Yaskawa INFORM job: A_ROOF_SIDE_0617_2_PAINT_25.JBI

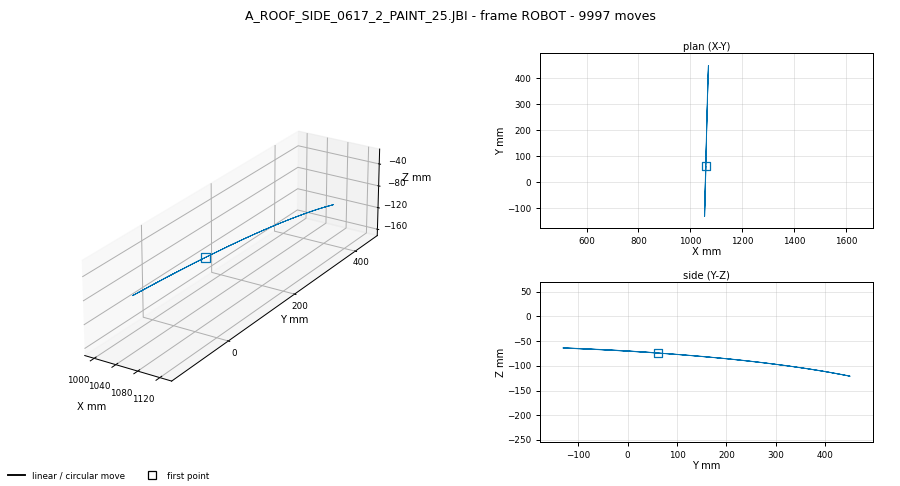
[picture p0: tool path of A_ROOF_SIDE_0617_2_PAINT_25.JBI in frame ROBOT, 9997 of 9997 moves have a stored position in this frame; points joined in program order, loops and branches not executed]
/JOB
//NAME A_ROOF_SIDE_0617_2_PAINT25
//POS
///NPOS 9997,0,0,0,0,0
///TOOL 1
///USER 0
///POSTYPE ROBOT
///RECTAN
///RCONF 1,0,0,0,0,0,0,0,0,0,0,0,0,0,0,0,0,0,0,0,0,0,0,0
C00000=1059.845,61.842,-73.709,171.756,29.525,155.487
C00001=1059.838,61.557,-73.690,171.754,29.522,155.486
C00002=1059.832,61.309,-73.673,171.753,29.519,155.486
C00003=1059.826,61.059,-73.655,171.752,29.517,155.485
C00004=1059.820,60.810,-73.638,171.750,29.515,155.485
C00005=1059.814,60.561,-73.621,171.748,29.512,155.485
C00006=1059.807,60.311,-73.604,171.747,29.509,155.484
C00007=1059.801,60.062,-73.587,171.746,29.507,155.484
C00008=1059.795,59.813,-73.569,171.744,29.505,155.484
C00009=1059.789,59.563,-73.553,171.743,29.502,155.483
C00010=1059.783,59.314,-73.535,171.741,29.500,155.483
C00011=1059.777,59.065,-73.518,171.739,29.497,155.482
C00012=1059.771,58.816,-73.501,171.739,29.494,155.482
C00013=1059.765,58.566,-73.483,171.737,29.492,155.482
C00014=1059.758,58.317,-73.466,171.735,29.489,155.481
C00015=1059.752,58.067,-73.450,171.733,29.487,155.481
C00016=1059.746,57.818,-73.432,171.733,29.485,155.481
C00017=1059.740,57.569,-73.415,171.731,29.482,155.480
C00018=1059.734,57.319,-73.398,171.729,29.479,155.480
C00019=1059.728,57.070,-73.381,171.728,29.477,155.480
C00020=1059.722,56.821,-73.365,171.726,29.474,155.479
C00021=1059.716,56.571,-73.347,171.725,29.472,155.479
C00022=1059.710,56.322,-73.330,171.723,29.470,155.478
C00023=1059.703,56.072,-73.313,171.722,29.467,155.478
C00024=1059.698,55.823,-73.296,171.720,29.464,155.478
C00025=1059.692,55.574,-73.279,171.719,29.462,155.477
C00026=1059.685,55.324,-73.262,171.718,29.459,155.477
C00027=1059.680,55.075,-73.245,171.716,29.457,155.477
C00028=1059.673,54.826,-73.228,171.714,29.454,155.476
C00029=1059.666,54.577,-73.211,171.712,29.452,155.476
C00030=1059.661,54.327,-73.194,171.712,29.449,155.475
C00031=1059.655,54.078,-73.177,171.710,29.446,155.475
C00032=1059.648,53.828,-73.161,171.708,29.444,155.475
C00033=1059.643,53.579,-73.143,171.707,29.441,155.474
C00034=1059.637,53.330,-73.127,171.706,29.439,155.474
C00035=1059.631,53.081,-73.110,171.704,29.437,155.474
C00036=1059.625,52.831,-73.093,171.703,29.434,155.473
C00037=1059.619,52.582,-73.076,171.701,29.431,155.473
C00038=1059.613,52.333,-73.059,171.700,29.429,155.473
C00039=1059.607,52.083,-73.041,171.698,29.426,155.472
C00040=1059.601,51.834,-73.025,171.697,29.424,155.472
C00041=1059.595,51.584,-73.009,171.695,29.422,155.472
C00042=1059.589,51.335,-72.991,171.693,29.419,155.471
C00043=1059.583,51.085,-72.975,171.693,29.416,155.471
C00044=1059.576,50.836,-72.958,171.691,29.413,155.470
C00045=1059.571,50.587,-72.941,171.689,29.411,155.470
C00046=1059.565,50.338,-72.924,171.688,29.409,155.470
C00047=1059.558,50.088,-72.907,171.687,29.406,155.469
C00048=1059.553,49.838,-72.890,171.685,29.404,155.469
C00049=1059.547,49.590,-72.873,171.683,29.401,155.469
C00050=1059.541,49.340,-72.857,171.682,29.398,155.468
C00051=1059.534,49.091,-72.840,171.680,29.396,155.468
C00052=1059.529,48.841,-72.823,171.679,29.394,155.467
C00053=1059.523,48.592,-72.807,171.678,29.391,155.467
C00054=1059.517,48.343,-72.790,171.676,29.388,155.467
C00055=1059.511,48.093,-72.773,171.674,29.386,155.466
C00056=1059.505,47.843,-72.756,171.674,29.383,155.466
C00057=1059.499,47.595,-72.739,171.672,29.381,155.466
C00058=1059.493,47.345,-72.723,171.670,29.378,155.465
C00059=1059.487,47.096,-72.706,171.668,29.376,155.465
C00060=1059.481,46.847,-72.689,171.668,29.373,155.464
C00061=1059.475,46.597,-72.673,171.666,29.370,155.464
C00062=1059.468,46.313,-72.654,171.664,29.368,155.464
C00063=1059.462,46.027,-72.634,171.663,29.365,155.463
C00064=1059.455,45.742,-72.615,171.661,29.361,155.463
C00065=1059.448,45.458,-72.596,171.659,29.359,155.462
C00066=1059.442,45.208,-72.580,171.658,29.356,155.462
C00067=1059.436,44.959,-72.563,171.656,29.354,155.462
C00068=1059.430,44.709,-72.547,171.654,29.351,155.461
C00069=1059.424,44.461,-72.530,171.654,29.348,155.461
C00070=1059.419,44.211,-72.513,171.652,29.346,155.461
C00071=1059.412,43.961,-72.497,171.650,29.343,155.460
C00072=1059.406,43.711,-72.480,171.649,29.341,155.460
C00073=1059.401,43.462,-72.464,171.648,29.338,155.459
C00074=1059.394,43.213,-72.447,171.646,29.336,155.459
C00075=1059.388,42.964,-72.431,171.645,29.333,155.459
C00076=1059.382,42.715,-72.415,171.643,29.331,155.458
C00077=1059.376,42.465,-72.398,171.641,29.328,155.458
C00078=1059.370,42.215,-72.382,171.640,29.326,155.458
C00079=1059.364,41.966,-72.365,171.639,29.324,155.457
C00080=1059.358,41.717,-72.349,171.637,29.321,155.457
C00081=1059.352,41.468,-72.332,171.635,29.319,155.457
C00082=1059.346,41.218,-72.316,171.635,29.316,155.456
C00083=1059.340,40.969,-72.300,171.633,29.313,155.456
C00084=1059.333,40.719,-72.283,171.631,29.311,155.455
C00085=1059.327,40.470,-72.267,171.630,29.308,155.455
C00086=1059.322,40.220,-72.250,171.628,29.306,155.455
C00087=1059.316,39.971,-72.234,171.627,29.304,155.454
C00088=1059.310,39.721,-72.217,171.625,29.301,155.454
C00089=1059.304,39.472,-72.201,171.624,29.299,155.454
C00090=1059.298,39.223,-72.185,171.622,29.296,155.453
C00091=1059.292,38.973,-72.169,171.620,29.293,155.453
C00092=1059.286,38.724,-72.152,171.620,29.291,155.453
C00093=1059.280,38.474,-72.136,171.618,29.288,155.452
C00094=1059.274,38.225,-72.120,171.616,29.286,155.452
C00095=1059.268,37.975,-72.103,171.615,29.283,155.452
C00096=1059.262,37.726,-72.087,171.614,29.281,155.451
C00097=1059.255,37.477,-72.071,171.612,29.279,155.451
C00098=1059.249,37.228,-72.055,171.610,29.276,155.450
C00099=1059.243,36.978,-72.039,171.609,29.274,155.450
C00100=1059.237,36.729,-72.023,171.607,29.271,155.450
C00101=1059.231,36.479,-72.006,171.606,29.269,155.449
C00102=1059.224,36.230,-71.990,171.605,29.266,155.449
C00103=1059.218,35.980,-71.974,171.603,29.264,155.449
C00104=1059.212,35.731,-71.958,171.601,29.261,155.448
C00105=1059.206,35.482,-71.942,171.600,29.259,155.448
C00106=1059.200,35.232,-71.925,171.599,29.256,155.448
C00107=1059.194,34.983,-71.910,171.597,29.254,155.447
C00108=1059.188,34.734,-71.893,171.595,29.252,155.447
C00109=1059.182,34.484,-71.878,171.594,29.249,155.447
C00110=1059.176,34.235,-71.862,171.593,29.247,155.446
C00111=1059.170,33.985,-71.845,171.591,29.244,155.446
C00112=1059.164,33.736,-71.830,171.590,29.242,155.446
C00113=1059.158,33.487,-71.813,171.588,29.239,155.445
C00114=1059.152,33.238,-71.797,171.586,29.237,155.445
C00115=1059.146,32.988,-71.781,171.586,29.234,155.445
C00116=1059.139,32.738,-71.765,171.584,29.232,155.444
C00117=1059.133,32.488,-71.749,171.582,29.229,155.444
C00118=1059.127,32.239,-71.733,171.580,29.227,155.444
C00119=1059.121,31.990,-71.717,171.579,29.224,155.443
C00120=1059.115,31.740,-71.701,171.578,29.222,155.443
C00121=1059.108,31.491,-71.686,171.576,29.220,155.443
C00122=1059.103,31.241,-71.669,171.575,29.217,155.442
C00123=1059.097,30.992,-71.653,171.573,29.215,155.442
C00124=1059.091,30.743,-71.637,171.571,29.212,155.442
C00125=1059.085,30.493,-71.621,171.571,29.210,155.441
C00126=1059.078,30.209,-71.603,171.569,29.207,155.441
C00127=1059.071,29.923,-71.585,171.567,29.204,155.440
C00128=1059.064,29.639,-71.566,171.565,29.201,155.440
C00129=1059.057,29.354,-71.549,171.563,29.199,155.440
C00130=1059.051,29.105,-71.532,171.562,29.196,155.439
C00131=1059.045,28.855,-71.517,171.561,29.194,155.439
C00132=1059.039,28.606,-71.501,171.559,29.191,155.439
C00133=1059.033,28.356,-71.485,171.557,29.189,155.438
C00134=1059.027,28.106,-71.469,171.556,29.186,155.438
C00135=1059.020,27.857,-71.454,171.555,29.184,155.438
C00136=1059.014,27.608,-71.438,171.553,29.181,155.437
C00137=1059.009,27.358,-71.422,171.551,29.179,155.437
C00138=1059.002,27.109,-71.406,171.550,29.177,155.437
C00139=1058.996,26.860,-71.390,171.548,29.174,155.436
C00140=1058.990,26.610,-71.375,171.547,29.172,155.436
C00141=1058.984,26.361,-71.359,171.546,29.169,155.436
C00142=1058.977,26.111,-71.343,171.544,29.167,155.435
C00143=1058.971,25.862,-71.328,171.542,29.164,155.435
C00144=1058.965,25.612,-71.311,171.541,29.162,155.435
C00145=1058.959,25.363,-71.296,171.540,29.160,155.434
C00146=1058.953,25.113,-71.280,171.538,29.158,155.434
C00147=1058.946,24.864,-71.265,171.536,29.155,155.434
C00148=1058.941,24.614,-71.249,171.535,29.153,155.433
C00149=1058.935,24.366,-71.234,171.533,29.150,155.433
C00150=1058.929,24.116,-71.218,171.532,29.148,155.432
C00151=1058.922,23.867,-71.203,171.531,29.146,155.432
C00152=1058.917,23.617,-71.187,171.529,29.143,155.432
C00153=1058.910,23.368,-71.171,171.527,29.141,155.432
C00154=1058.904,23.118,-71.156,171.526,29.138,155.431
C00155=1058.898,22.869,-71.140,171.525,29.136,155.431
C00156=1058.892,22.619,-71.125,171.523,29.134,155.431
C00157=1058.886,22.369,-71.108,171.522,29.131,155.430
C00158=1058.880,22.120,-71.093,171.520,29.129,155.430
C00159=1058.874,21.870,-71.077,171.518,29.126,155.430
C00160=1058.868,21.622,-71.063,171.517,29.124,155.429
C00161=1058.862,21.372,-71.046,171.516,29.122,155.429
C00162=1058.856,21.123,-71.031,171.514,29.119,155.429
C00163=1058.850,20.873,-71.015,171.512,29.117,155.428
C00164=1058.843,20.624,-71.000,171.511,29.114,155.428
C00165=1058.837,20.374,-70.984,171.509,29.112,155.428
C00166=1058.831,20.125,-70.969,171.508,29.109,155.427
C00167=1058.825,19.875,-70.954,171.507,29.107,155.427
C00168=1058.819,19.626,-70.938,171.505,29.105,155.427
C00169=1058.813,19.377,-70.923,171.503,29.102,155.426
C00170=1058.807,19.127,-70.907,171.502,29.100,155.426
C00171=1058.801,18.878,-70.892,171.501,29.098,155.426
C00172=1058.794,18.628,-70.877,171.499,29.095,155.425
C00173=1058.788,18.379,-70.861,171.497,29.093,155.425
C00174=1058.782,18.129,-70.846,171.496,29.090,155.425
C00175=1058.776,17.879,-70.830,171.494,29.088,155.424
C00176=1058.770,17.631,-70.815,171.493,29.086,155.424
C00177=1058.764,17.381,-70.800,171.492,29.083,155.424
C00178=1058.758,17.131,-70.784,171.490,29.081,155.423
C00179=1058.751,16.882,-70.769,171.488,29.079,155.423
C00180=1058.745,16.632,-70.754,171.487,29.076,155.423
C00181=1058.739,16.382,-70.738,171.485,29.074,155.422
C00182=1058.733,16.134,-70.723,171.484,29.071,155.422
C00183=1058.728,15.884,-70.707,171.482,29.069,155.422
C00184=1058.721,15.634,-70.693,171.481,29.067,155.421
C00185=1058.715,15.385,-70.678,171.479,29.064,155.421
C00186=1058.709,15.135,-70.661,171.477,29.062,155.421
C00187=1058.703,14.886,-70.647,171.477,29.060,155.420
C00188=1058.697,14.637,-70.632,171.475,29.057,155.420
C00189=1058.691,14.387,-70.616,171.473,29.055,155.420
C00190=1058.684,14.104,-70.599,171.472,29.052,155.419
C00191=1058.676,13.820,-70.581,171.470,29.050,155.419
C00192=1058.669,13.537,-70.565,171.468,29.047,155.419
C00193=1058.662,13.253,-70.547,171.467,29.044,155.418
C00194=1058.656,13.004,-70.532,171.465,29.042,155.418
C00195=1058.650,12.754,-70.517,171.463,29.040,155.418
C00196=1058.644,12.504,-70.502,171.462,29.037,155.417
C00197=1058.637,12.255,-70.487,171.460,29.035,155.417
C00198=1058.631,12.005,-70.472,171.458,29.033,155.417
C00199=1058.625,11.756,-70.457,171.457,29.031,155.417
C00200=1058.619,11.507,-70.442,171.456,29.028,155.416
C00201=1058.613,11.257,-70.427,171.454,29.026,155.416
C00202=1058.606,11.007,-70.412,171.452,29.023,155.416
C00203=1058.600,10.758,-70.397,171.451,29.021,155.415
C00204=1058.594,10.509,-70.382,171.449,29.019,155.415
C00205=1058.588,10.259,-70.367,171.447,29.016,155.415
C00206=1058.581,10.010,-70.352,171.447,29.014,155.414
C00207=1058.576,9.760,-70.337,171.445,29.012,155.414
C00208=1058.570,9.511,-70.322,171.443,29.010,155.414
C00209=1058.563,9.262,-70.307,171.442,29.007,155.413
C00210=1058.557,9.012,-70.292,171.440,29.005,155.413
C00211=1058.551,8.762,-70.277,171.438,29.003,155.413
C00212=1058.545,8.513,-70.262,171.437,29.001,155.413
C00213=1058.538,8.264,-70.247,171.436,28.999,155.412
C00214=1058.532,8.014,-70.232,171.434,28.996,155.412
C00215=1058.526,7.764,-70.217,171.432,28.994,155.412
C00216=1058.520,7.515,-70.203,171.431,28.991,155.411
C00217=1058.514,7.265,-70.187,171.429,28.989,155.411
C00218=1058.508,7.016,-70.172,171.428,28.987,155.411
C00219=1058.502,6.767,-70.158,171.427,28.984,155.410
C00220=1058.496,6.517,-70.143,171.425,28.982,155.410
C00221=1058.489,6.267,-70.128,171.423,28.980,155.410
C00222=1058.483,6.018,-70.113,171.421,28.978,155.410
C00223=1058.477,5.769,-70.098,171.420,28.975,155.409
C00224=1058.471,5.519,-70.083,171.418,28.973,155.409
C00225=1058.464,5.270,-70.068,171.417,28.971,155.409
C00226=1058.459,5.020,-70.054,171.416,28.969,155.408
C00227=1058.452,4.770,-70.039,171.414,28.966,155.408
C00228=1058.446,4.521,-70.024,171.412,28.964,155.408
C00229=1058.440,4.272,-70.010,171.411,28.961,155.407
C00230=1058.434,4.022,-69.995,171.409,28.959,155.407
C00231=1058.428,3.772,-69.979,171.408,28.957,155.407
C00232=1058.422,3.523,-69.965,171.407,28.954,155.406
C00233=1058.416,3.273,-69.950,171.405,28.952,155.406
C00234=1058.410,3.025,-69.935,171.403,28.950,155.406
C00235=1058.404,2.775,-69.920,171.401,28.948,155.406
C00236=1058.398,2.525,-69.906,171.400,28.945,155.405
C00237=1058.392,2.276,-69.892,171.398,28.943,155.405
C00238=1058.386,2.026,-69.877,171.397,28.941,155.405
C00239=1058.379,1.776,-69.862,171.396,28.939,155.404
C00240=1058.374,1.527,-69.847,171.394,28.936,155.404
C00241=1058.367,1.278,-69.832,171.392,28.934,155.404
C00242=1058.362,1.028,-69.818,171.391,28.931,155.403
C00243=1058.355,0.778,-69.803,171.389,28.929,155.403
C00244=1058.349,0.529,-69.788,171.387,28.927,155.403
C00245=1058.343,0.280,-69.774,171.386,28.925,155.403
C00246=1058.337,0.030,-69.759,171.385,28.922,155.402
C00247=1058.331,-0.219,-69.745,171.383,28.920,155.402
C00248=1058.325,-0.469,-69.730,171.381,28.918,155.402
C00249=1058.319,-0.718,-69.715,171.380,28.915,155.401
C00250=1058.313,-0.968,-69.701,171.378,28.913,155.401
C00251=1058.307,-1.217,-69.687,171.376,28.910,155.401
C00252=1058.301,-1.467,-69.672,171.376,28.908,155.400
C00253=1058.294,-1.717,-69.657,171.374,28.906,155.400
C00254=1058.288,-1.998,-69.640,171.372,28.903,155.400
C00255=1058.281,-2.280,-69.624,171.371,28.901,155.400
C00256=1058.275,-2.561,-69.608,171.368,28.898,155.399
C00257=1058.268,-2.843,-69.591,171.366,28.896,155.399
C00258=1058.262,-3.092,-69.577,171.365,28.893,155.398
C00259=1058.256,-3.342,-69.562,171.364,28.891,155.398
C00260=1058.250,-3.592,-69.548,171.362,28.889,155.398
C00261=1058.243,-3.841,-69.534,171.361,28.887,155.398
C00262=1058.237,-4.091,-69.519,171.359,28.885,155.397
C00263=1058.231,-4.340,-69.505,171.357,28.882,155.397
C00264=1058.225,-4.590,-69.490,171.356,28.880,155.397
C00265=1058.219,-4.839,-69.477,171.354,28.878,155.397
C00266=1058.212,-5.089,-69.462,171.352,28.876,155.396
C00267=1058.206,-5.339,-69.447,171.351,28.874,155.396
C00268=1058.200,-5.588,-69.433,171.350,28.872,155.396
C00269=1058.193,-5.837,-69.418,171.348,28.869,155.395
C00270=1058.188,-6.087,-69.405,171.346,28.867,155.395
C00271=1058.181,-6.336,-69.390,171.345,28.865,155.395
C00272=1058.175,-6.586,-69.376,171.343,28.863,155.395
C00273=1058.169,-6.835,-69.361,171.341,28.860,155.394
C00274=1058.163,-7.085,-69.348,171.339,28.858,155.394
C00275=1058.156,-7.334,-69.333,171.338,28.856,155.394
C00276=1058.151,-7.584,-69.319,171.337,28.854,155.394
C00277=1058.144,-7.834,-69.304,171.335,28.852,155.393
C00278=1058.138,-8.083,-69.291,171.334,28.850,155.393
C00279=1058.132,-8.332,-69.276,171.332,28.847,155.393
C00280=1058.126,-8.582,-69.262,171.330,28.845,155.392
C00281=1058.119,-8.831,-69.248,171.329,28.843,155.392
C00282=1058.114,-9.081,-69.234,171.327,28.841,155.392
C00283=1058.107,-9.331,-69.219,171.325,28.839,155.392
C00284=1058.102,-9.580,-69.205,171.323,28.836,155.391
C00285=1058.095,-9.830,-69.191,171.323,28.834,155.391
C00286=1058.089,-10.079,-69.177,171.321,28.832,155.391
C00287=1058.083,-10.329,-69.162,171.319,28.830,155.390
C00288=1058.077,-10.578,-69.149,171.318,28.828,155.390
C00289=1058.070,-10.828,-69.134,171.316,28.825,155.390
C00290=1058.065,-11.077,-69.120,171.314,28.823,155.390
C00291=1058.058,-11.327,-69.106,171.313,28.821,155.389
C00292=1058.052,-11.576,-69.092,171.311,28.819,155.389
C00293=1058.047,-11.826,-69.078,171.309,28.817,155.389
C00294=1058.040,-12.075,-69.064,171.308,28.815,155.389
C00295=1058.034,-12.325,-69.050,171.307,28.812,155.388
C00296=1058.027,-12.575,-69.036,171.305,28.810,155.388
C00297=1058.021,-12.824,-69.022,171.303,28.808,155.388
C00298=1058.016,-13.073,-69.008,171.302,28.806,155.387
C00299=1058.009,-13.323,-68.994,171.300,28.804,155.387
C00300=1058.003,-13.572,-68.979,171.298,28.801,155.387
C00301=1057.997,-13.822,-68.965,171.297,28.799,155.387
C00302=1057.991,-14.072,-68.952,171.295,28.797,155.387
C00303=1057.985,-14.321,-68.937,171.293,28.795,155.386
C00304=1057.979,-14.571,-68.923,171.292,28.793,155.386
C00305=1057.973,-14.820,-68.910,171.291,28.791,155.386
C00306=1057.967,-15.070,-68.895,171.289,28.789,155.385
C00307=1057.960,-15.319,-68.882,171.287,28.787,155.385
C00308=1057.955,-15.569,-68.868,171.286,28.784,155.385
C00309=1057.948,-15.819,-68.854,171.284,28.782,155.385
C00310=1057.942,-16.068,-68.840,171.282,28.780,155.384
C00311=1057.936,-16.318,-68.826,171.281,28.778,155.384
C00312=1057.929,-16.567,-68.813,171.279,28.776,155.384
C00313=1057.923,-16.817,-68.798,171.277,28.774,155.384
C00314=1057.917,-17.066,-68.785,171.275,28.772,155.383
C00315=1057.911,-17.315,-68.771,171.275,28.770,155.383
C00316=1057.904,-17.565,-68.757,171.273,28.767,155.383
C00317=1057.899,-17.815,-68.743,171.271,28.766,155.383
C00318=1057.893,-18.069,-68.729,171.270,28.764,155.382
C00319=1057.886,-18.325,-68.715,171.268,28.761,155.382
C00320=1057.879,-18.579,-68.701,171.266,28.759,155.382
C00321=1057.873,-18.833,-68.687,171.265,28.757,155.382
C00322=1057.867,-19.083,-68.674,171.263,28.755,155.381
C00323=1057.861,-19.333,-68.659,171.261,28.753,155.381
C00324=1057.855,-19.582,-68.646,171.259,28.751,155.381
C00325=1057.849,-19.832,-68.632,171.258,28.749,155.381
C00326=1057.842,-20.082,-68.619,171.256,28.746,155.380
C00327=1057.836,-20.331,-68.605,171.254,28.744,155.380
C00328=1057.830,-20.580,-68.591,171.253,28.743,155.380
C00329=1057.824,-20.830,-68.577,171.251,28.740,155.380
C00330=1057.818,-21.079,-68.563,171.250,28.738,155.379
C00331=1057.812,-21.329,-68.550,171.248,28.736,155.379
C00332=1057.805,-21.579,-68.536,171.247,28.734,155.379
C00333=1057.800,-21.828,-68.522,171.245,28.732,155.379
C00334=1057.793,-22.078,-68.509,171.243,28.730,155.378
C00335=1057.787,-22.328,-68.496,171.242,28.728,155.378
C00336=1057.781,-22.577,-68.482,171.240,28.726,155.378
C00337=1057.775,-22.826,-68.468,171.238,28.724,155.378
C00338=1057.769,-23.076,-68.455,171.236,28.722,155.377
C00339=1057.763,-23.326,-68.441,171.235,28.719,155.377
C00340=1057.756,-23.575,-68.428,171.233,28.717,155.377
C00341=1057.751,-23.825,-68.414,171.231,28.715,155.377
C00342=1057.745,-24.074,-68.401,171.230,28.713,155.376
C00343=1057.738,-24.324,-68.387,171.228,28.711,155.376
C00344=1057.732,-24.574,-68.373,171.226,28.709,155.376
C00345=1057.726,-24.823,-68.360,171.226,28.707,155.376
C00346=1057.720,-25.072,-68.346,171.224,28.705,155.375
C00347=1057.714,-25.322,-68.332,171.222,28.703,155.375
C00348=1057.708,-25.572,-68.319,171.220,28.701,155.375
C00349=1057.701,-25.821,-68.306,171.219,28.699,155.375
C00350=1057.696,-26.070,-68.292,171.217,28.697,155.375
C00351=1057.689,-26.320,-68.278,171.215,28.695,155.374
C00352=1057.683,-26.570,-68.265,171.214,28.693,155.374
C00353=1057.677,-26.819,-68.251,171.212,28.690,155.374
C00354=1057.671,-27.069,-68.238,171.210,28.689,155.374
C00355=1057.665,-27.318,-68.225,171.208,28.686,155.373
C00356=1057.659,-27.568,-68.212,171.207,28.685,155.373
C00357=1057.652,-27.818,-68.198,171.205,28.683,155.373
C00358=1057.646,-28.067,-68.185,171.203,28.680,155.373
C00359=1057.640,-28.316,-68.172,171.202,28.679,155.372
C00360=1057.634,-28.566,-68.158,171.200,28.677,155.372
C00361=1057.628,-28.816,-68.145,171.198,28.675,155.372
C00362=1057.621,-29.090,-68.130,171.196,28.673,155.372
C00363=1057.614,-29.365,-68.115,171.195,28.670,155.372
C00364=1057.607,-29.640,-68.101,171.193,28.668,155.371
C00365=1057.599,-29.916,-68.086,171.191,28.666,155.371
C00366=1057.594,-30.166,-68.073,171.190,28.664,155.371
C00367=1057.588,-30.415,-68.060,171.188,28.662,155.371
C00368=1057.582,-30.664,-68.047,171.186,28.660,155.370
C00369=1057.576,-30.914,-68.033,171.185,28.658,155.370
C00370=1057.569,-31.164,-68.020,171.183,28.656,155.370
C00371=1057.563,-31.413,-68.007,171.181,28.654,155.370
C00372=1057.557,-31.663,-67.994,171.179,28.652,155.369
C00373=1057.550,-31.912,-67.981,171.178,28.651,155.369
C00374=1057.545,-32.162,-67.968,171.176,28.648,155.369
C00375=1057.538,-32.411,-67.955,171.174,28.647,155.369
C00376=1057.532,-32.661,-67.941,171.173,28.644,155.369
C00377=1057.526,-32.911,-67.927,171.171,28.642,155.368
C00378=1057.520,-33.161,-67.915,171.169,28.641,155.368
C00379=1057.514,-33.410,-67.901,171.167,28.638,155.368
C00380=1057.508,-33.659,-67.888,171.166,28.637,155.368
C00381=1057.502,-33.909,-67.876,171.164,28.634,155.368
C00382=1057.494,-34.188,-67.860,171.162,28.632,155.367
C00383=1057.487,-34.467,-67.846,171.161,28.631,155.367
C00384=1057.481,-34.747,-67.832,171.159,28.628,155.367
C00385=1057.474,-35.026,-67.817,171.157,28.626,155.367
C00386=1057.468,-35.275,-67.804,171.156,28.624,155.366
C00387=1057.461,-35.525,-67.791,171.154,28.622,155.366
C00388=1057.455,-35.775,-67.777,171.152,28.620,155.366
C00389=1057.449,-36.025,-67.765,171.150,28.618,155.366
C00390=1057.443,-36.274,-67.752,171.149,28.616,155.365
C00391=1057.437,-36.524,-67.739,171.147,28.615,155.365
C00392=1057.431,-36.773,-67.726,171.145,28.612,155.365
C00393=1057.425,-37.022,-67.712,171.143,28.611,155.365
C00394=1057.419,-37.272,-67.700,171.142,28.608,155.365
C00395=1057.413,-37.522,-67.686,171.140,28.607,155.364
C00396=1057.407,-37.772,-67.673,171.138,28.605,155.364
C00397=1057.401,-38.021,-67.660,171.137,28.603,155.364
C00398=1057.395,-38.271,-67.648,171.135,28.601,155.364
C00399=1057.389,-38.520,-67.634,171.133,28.599,155.364
C00400=1057.383,-38.770,-67.622,171.131,28.597,155.363
C00401=1057.376,-39.020,-67.609,171.130,28.595,155.363
C00402=1057.370,-39.269,-67.596,171.128,28.594,155.363
C00403=1057.363,-39.519,-67.583,171.126,28.591,155.363
C00404=1057.357,-39.769,-67.570,171.125,28.590,155.363
C00405=1057.351,-40.018,-67.557,171.123,28.588,155.362
C00406=1057.345,-40.267,-67.545,171.121,28.586,155.362
C00407=1057.338,-40.517,-67.532,171.119,28.584,155.362
C00408=1057.333,-40.767,-67.519,171.118,28.583,155.362
C00409=1057.327,-41.016,-67.507,171.116,28.580,155.362
C00410=1057.320,-41.266,-67.494,171.114,28.579,155.362
C00411=1057.314,-41.516,-67.481,171.112,28.577,155.361
C00412=1057.308,-41.765,-67.468,171.111,28.575,155.361
C00413=1057.302,-42.014,-67.456,171.109,28.573,155.361
C00414=1057.296,-42.264,-67.443,171.107,28.571,155.361
C00415=1057.289,-42.514,-67.430,171.106,28.569,155.361
C00416=1057.284,-42.763,-67.417,171.104,28.568,155.360
C00417=1057.277,-43.012,-67.405,171.102,28.566,155.360
C00418=1057.271,-43.262,-67.392,171.100,28.564,155.360
C00419=1057.265,-43.512,-67.380,171.099,28.562,155.360
C00420=1057.259,-43.761,-67.366,171.097,28.560,155.360
C00421=1057.252,-44.011,-67.354,171.095,28.558,155.359
C00422=1057.246,-44.261,-67.342,171.093,28.557,155.359
C00423=1057.240,-44.510,-67.329,171.092,28.555,155.359
C00424=1057.234,-44.760,-67.316,171.090,28.553,155.359
C00425=1057.228,-45.010,-67.303,171.088,28.551,155.359
C00426=1057.221,-45.259,-67.291,171.087,28.549,155.359
C00427=1057.215,-45.509,-67.278,171.085,28.548,155.358
C00428=1057.209,-45.759,-67.266,171.083,28.546,155.358
C00429=1057.203,-46.009,-67.253,171.081,28.544,155.358
C00430=1057.196,-46.257,-67.240,171.080,28.542,155.358
C00431=1057.190,-46.507,-67.228,171.078,28.541,155.358
C00432=1057.185,-46.757,-67.215,171.076,28.538,155.357
C00433=1057.179,-47.007,-67.203,171.074,28.537,155.357
C00434=1057.172,-47.256,-67.190,171.073,28.535,155.357
C00435=1057.166,-47.506,-67.177,171.071,28.533,155.357
C00436=1057.160,-47.756,-67.165,171.069,28.531,155.357
C00437=1057.154,-48.006,-67.152,171.067,28.530,155.357
C00438=1057.147,-48.255,-67.140,171.066,28.528,155.356
C00439=1057.142,-48.504,-67.128,171.064,28.526,155.356
C00440=1057.136,-48.754,-67.115,171.062,28.524,155.356
C00441=1057.130,-49.004,-67.102,171.061,28.522,155.356
C00442=1057.123,-49.253,-67.090,171.059,28.521,155.356
C00443=1057.117,-49.503,-67.078,171.057,28.519,155.356
C00444=1057.111,-49.752,-67.065,171.055,28.517,155.355
C00445=1057.104,-50.002,-67.053,171.054,28.515,155.355
C00446=1057.098,-50.282,-67.039,171.052,28.514,155.355
C00447=1057.091,-50.561,-67.025,171.050,28.511,155.355
C00448=1057.084,-50.842,-67.011,171.047,28.509,155.355
C00449=1057.077,-51.121,-66.997,171.046,28.508,155.354
C00450=1057.071,-51.370,-66.985,171.044,28.506,155.354
C00451=1057.065,-51.620,-66.973,171.042,28.505,155.354
C00452=1057.058,-51.870,-66.961,171.040,28.503,155.354
C00453=1057.052,-52.120,-66.948,171.039,28.501,155.354
C00454=1057.045,-52.369,-66.936,171.037,28.500,155.354
C00455=1057.039,-52.619,-66.924,171.035,28.498,155.354
C00456=1057.033,-52.869,-66.912,171.033,28.496,155.353
C00457=1057.026,-53.118,-66.900,171.032,28.495,155.353
C00458=1057.021,-53.367,-66.888,171.030,28.493,155.353
C00459=1057.014,-53.617,-66.876,171.028,28.491,155.353
C00460=1057.008,-53.867,-66.863,171.027,28.490,155.353
C00461=1057.002,-54.116,-66.851,171.025,28.488,155.353
C00462=1056.995,-54.366,-66.839,171.023,28.486,155.353
C00463=1056.989,-54.616,-66.827,171.021,28.485,155.352
C00464=1056.982,-54.865,-66.815,171.020,28.483,155.352
C00465=1056.977,-55.115,-66.802,171.018,28.481,155.352
C00466=1056.971,-55.364,-66.791,171.015,28.480,155.352
C00467=1056.964,-55.614,-66.779,171.013,28.478,155.352
C00468=1056.958,-55.864,-66.766,171.012,28.476,155.352
C00469=1056.951,-56.113,-66.754,171.010,28.475,155.352
C00470=1056.945,-56.363,-66.742,171.008,28.473,155.351
C00471=1056.939,-56.613,-66.730,171.006,28.471,155.351
C00472=1056.932,-56.862,-66.718,171.005,28.470,155.351
C00473=1056.927,-57.111,-66.705,171.003,28.468,155.351
C00474=1056.920,-57.361,-66.693,171.001,28.466,155.351
C00475=1056.914,-57.611,-66.682,170.999,28.465,155.351
C00476=1056.908,-57.861,-66.670,170.997,28.464,155.351
C00477=1056.901,-58.111,-66.658,170.996,28.462,155.350
C00478=1056.895,-58.360,-66.646,170.994,28.460,155.350
C00479=1056.889,-58.609,-66.634,170.992,28.459,155.350
C00480=1056.883,-58.859,-66.622,170.990,28.457,155.350
C00481=1056.877,-59.109,-66.609,170.989,28.455,155.350
C00482=1056.870,-59.358,-66.597,170.987,28.454,155.350
C00483=1056.864,-59.608,-66.586,170.985,28.452,155.350
C00484=1056.858,-59.858,-66.574,170.984,28.451,155.349
C00485=1056.852,-60.107,-66.562,170.982,28.449,155.349
C00486=1056.845,-60.357,-66.550,170.980,28.448,155.349
C00487=1056.840,-60.606,-66.538,170.978,28.446,155.349
C00488=1056.834,-60.856,-66.526,170.976,28.445,155.349
C00489=1056.827,-61.106,-66.514,170.975,28.443,155.349
C00490=1056.821,-61.356,-66.502,170.972,28.441,155.349
C00491=1056.815,-61.605,-66.490,170.970,28.439,155.349
C00492=1056.809,-61.855,-66.479,170.969,28.438,155.348
C00493=1056.803,-62.105,-66.466,170.967,28.436,155.348
C00494=1056.796,-62.354,-66.454,170.965,28.435,155.348
C00495=1056.790,-62.603,-66.443,170.963,28.433,155.348
C00496=1056.784,-62.854,-66.431,170.961,28.432,155.348
C00497=1056.778,-63.103,-66.419,170.960,28.430,155.348
C00498=1056.771,-63.353,-66.407,170.958,28.428,155.348
C00499=1056.765,-63.602,-66.396,170.956,28.427,155.347
C00500=1056.759,-63.852,-66.384,170.954,28.426,155.347
C00501=1056.753,-64.102,-66.372,170.953,28.424,155.347
C00502=1056.747,-64.351,-66.360,170.951,28.422,155.347
C00503=1056.741,-64.601,-66.348,170.949,28.421,155.347
C00504=1056.735,-64.851,-66.336,170.947,28.419,155.347
C00505=1056.728,-65.100,-66.325,170.946,28.418,155.347
C00506=1056.723,-65.350,-66.313,170.944,28.416,155.347
C00507=1056.716,-65.600,-66.301,170.942,28.415,155.347
C00508=1056.710,-65.849,-66.290,170.940,28.413,155.346
C00509=1056.704,-66.099,-66.278,170.938,28.411,155.346
C00510=1056.697,-66.380,-66.265,170.936,28.410,155.346
C00511=1056.690,-66.660,-66.251,170.934,28.408,155.346
C00512=1056.683,-66.942,-66.238,170.932,28.406,155.346
C00513=1056.676,-67.223,-66.225,170.930,28.404,155.346
C00514=1056.671,-67.472,-66.213,170.928,28.403,155.346
C00515=1056.665,-67.722,-66.202,170.926,28.402,155.346
C00516=1056.658,-67.972,-66.190,170.924,28.400,155.345
C00517=1056.652,-68.221,-66.179,170.923,28.398,155.345
C00518=1056.646,-68.471,-66.166,170.921,28.397,155.345
C00519=1056.641,-68.721,-66.155,170.919,28.396,155.345
C00520=1056.634,-68.970,-66.144,170.917,28.394,155.345
C00521=1056.628,-69.220,-66.132,170.916,28.392,155.345
C00522=1056.622,-69.470,-66.120,170.914,28.391,155.345
C00523=1056.616,-69.720,-66.109,170.912,28.390,155.345
C00524=1056.610,-69.969,-66.097,170.910,28.388,155.344
C00525=1056.604,-70.219,-66.086,170.909,28.386,155.344
C00526=1056.598,-70.468,-66.074,170.906,28.385,155.344
C00527=1056.592,-70.718,-66.063,170.904,28.383,155.344
C00528=1056.586,-70.967,-66.051,170.902,28.382,155.344
C00529=1056.580,-71.217,-66.040,170.900,28.381,155.344
C00530=1056.574,-71.467,-66.027,170.899,28.379,155.344
C00531=1056.568,-71.717,-66.016,170.897,28.377,155.344
C00532=1056.561,-71.966,-66.004,170.895,28.376,155.344
C00533=1056.555,-72.216,-65.993,170.893,28.375,155.344
C00534=1056.549,-72.465,-65.982,170.892,28.373,155.343
C00535=1056.544,-72.715,-65.970,170.890,28.371,155.343
C00536=1056.537,-72.965,-65.959,170.888,28.370,155.343
C00537=1056.531,-73.214,-65.947,170.886,28.369,155.343
C00538=1056.525,-73.464,-65.936,170.885,28.367,155.343
C00539=1056.519,-73.714,-65.925,170.883,28.366,155.343
C00540=1056.513,-73.964,-65.913,170.881,28.364,155.343
C00541=1056.508,-74.213,-65.902,170.878,28.363,155.343
C00542=1056.501,-74.463,-65.890,170.876,28.361,155.343
C00543=1056.495,-74.712,-65.879,170.875,28.360,155.343
C00544=1056.489,-74.962,-65.868,170.873,28.359,155.342
C00545=1056.482,-75.212,-65.856,170.871,28.358,155.342
C00546=1056.477,-75.462,-65.845,170.869,28.356,155.342
C00547=1056.470,-75.712,-65.833,170.868,28.355,155.342
C00548=1056.465,-75.961,-65.823,170.866,28.353,155.342
C00549=1056.458,-76.211,-65.811,170.864,28.352,155.342
C00550=1056.451,-76.460,-65.800,170.862,28.350,155.342
C00551=1056.445,-76.710,-65.789,170.860,28.349,155.342
C00552=1056.439,-76.959,-65.778,170.859,28.348,155.342
C00553=1056.433,-77.209,-65.766,170.857,28.347,155.342
C00554=1056.427,-77.459,-65.755,170.854,28.345,155.342
C00555=1056.421,-77.709,-65.744,170.852,28.344,155.342
C00556=1056.415,-77.958,-65.733,170.851,28.342,155.341
C00557=1056.408,-78.208,-65.721,170.849,28.341,155.341
C00558=1056.402,-78.457,-65.710,170.847,28.340,155.341
C00559=1056.396,-78.708,-65.699,170.845,28.338,155.341
C00560=1056.390,-78.957,-65.688,170.843,28.337,155.341
C00561=1056.384,-79.206,-65.677,170.842,28.336,155.341
C00562=1056.378,-79.456,-65.665,170.840,28.335,155.341
C00563=1056.372,-79.706,-65.655,170.838,28.334,155.341
C00564=1056.366,-79.956,-65.643,170.836,28.332,155.341
C00565=1056.359,-80.205,-65.633,170.833,28.331,155.341
C00566=1056.353,-80.455,-65.622,170.832,28.330,155.341
C00567=1056.347,-80.704,-65.610,170.830,28.328,155.341
C00568=1056.341,-80.954,-65.599,170.828,28.327,155.341
C00569=1056.334,-81.203,-65.589,170.826,28.326,155.341
C00570=1056.328,-81.454,-65.577,170.824,28.325,155.341
C00571=1056.322,-81.703,-65.567,170.823,28.323,155.340
C00572=1056.316,-81.953,-65.555,170.821,28.322,155.340
C00573=1056.309,-82.203,-65.545,170.819,28.321,155.340
C00574=1056.302,-82.487,-65.532,170.816,28.320,155.340
C00575=1056.295,-82.769,-65.520,170.815,28.318,155.340
C00576=1056.288,-83.052,-65.508,170.813,28.317,155.340
C00577=1056.281,-83.336,-65.495,170.810,28.315,155.340
C00578=1056.275,-83.585,-65.484,170.808,28.314,155.340
C00579=1056.268,-83.835,-65.473,170.806,28.313,155.340
C00580=1056.263,-84.084,-65.462,170.805,28.312,155.340
C00581=1056.256,-84.334,-65.452,170.803,28.311,155.340
C00582=1056.250,-84.584,-65.440,170.801,28.309,155.340
C00583=1056.244,-84.833,-65.430,170.799,28.308,155.340
C00584=1056.237,-85.083,-65.419,170.796,28.307,155.340
C00585=1056.231,-85.333,-65.408,170.795,28.306,155.340
C00586=1056.225,-85.582,-65.397,170.793,28.305,155.340
C00587=1056.219,-85.832,-65.386,170.791,28.304,155.340
C00588=1056.213,-86.082,-65.376,170.789,28.302,155.340
C00589=1056.207,-86.332,-65.365,170.787,28.301,155.340
C00590=1056.201,-86.582,-65.354,170.786,28.300,155.339
C00591=1056.194,-86.831,-65.344,170.784,28.299,155.339
C00592=1056.188,-87.081,-65.333,170.782,28.298,155.339
C00593=1056.182,-87.331,-65.322,170.780,28.297,155.339
C00594=1056.176,-87.580,-65.312,170.777,28.295,155.339
C00595=1056.169,-87.830,-65.300,170.776,28.294,155.339
C00596=1056.164,-88.080,-65.289,170.774,28.293,155.339
C00597=1056.157,-88.329,-65.279,170.772,28.292,155.339
C00598=1056.151,-88.579,-65.268,170.770,28.291,155.339
C00599=1056.145,-88.828,-65.257,170.768,28.289,155.339
C00600=1056.139,-89.078,-65.247,170.766,28.288,155.339
C00601=1056.133,-89.328,-65.236,170.765,28.287,155.339
C00602=1056.127,-89.578,-65.225,170.763,28.286,155.339
C00603=1056.120,-89.827,-65.215,170.760,28.285,155.339
C00604=1056.114,-90.077,-65.204,170.758,28.284,155.339
C00605=1056.108,-90.326,-65.194,170.756,28.283,155.339
C00606=1056.102,-90.576,-65.183,170.755,28.281,155.339
C00607=1056.096,-90.827,-65.172,170.753,28.280,155.339
C00608=1056.089,-91.076,-65.162,170.751,28.279,155.339
C00609=1056.084,-91.325,-65.151,170.749,28.278,155.339
C00610=1056.078,-91.575,-65.140,170.747,28.277,155.339
C00611=1056.071,-91.825,-65.129,170.746,28.276,155.339
C00612=1056.065,-92.075,-65.119,170.744,28.275,155.339
C00613=1056.060,-92.324,-65.108,170.741,28.274,155.339
C00614=1056.053,-92.574,-65.098,170.739,28.273,155.339
C00615=1056.047,-92.824,-65.087,170.737,28.271,155.339
C00616=1056.041,-93.074,-65.077,170.735,28.270,155.339
C00617=1056.035,-93.323,-65.066,170.734,28.269,155.339
C00618=1056.029,-93.573,-65.056,170.732,28.268,155.339
C00619=1056.022,-93.822,-65.045,170.730,28.267,155.339
C00620=1056.017,-94.073,-65.035,170.728,28.266,155.338
C00621=1056.010,-94.322,-65.024,170.726,28.265,155.338
C00622=1056.004,-94.571,-65.014,170.724,28.264,155.338
C00623=1055.999,-94.821,-65.003,170.722,28.263,155.338
C00624=1055.992,-95.071,-64.993,170.720,28.262,155.338
C00625=1055.986,-95.321,-64.982,170.718,28.261,155.338
C00626=1055.980,-95.570,-64.972,170.716,28.260,155.338
C00627=1055.974,-95.820,-64.961,170.714,28.258,155.338
C00628=1055.968,-96.069,-64.951,170.713,28.257,155.338
C00629=1055.962,-96.320,-64.941,170.711,28.256,155.338
C00630=1055.956,-96.569,-64.930,170.709,28.255,155.338
C00631=1055.949,-96.819,-64.919,170.706,28.254,155.338
C00632=1055.944,-97.069,-64.909,170.704,28.253,155.338
C00633=1055.938,-97.318,-64.899,170.703,28.252,155.338
C00634=1055.931,-97.568,-64.888,170.701,28.251,155.338
C00635=1055.925,-97.818,-64.878,170.699,28.250,155.338
C00636=1055.919,-98.067,-64.867,170.697,28.249,155.338
C00637=1055.913,-98.317,-64.858,170.695,28.248,155.338
C00638=1055.906,-98.603,-64.845,170.692,28.247,155.338
C00639=1055.899,-98.888,-64.834,170.691,28.246,155.338
C00640=1055.892,-99.173,-64.822,170.688,28.245,155.338
C00641=1055.885,-99.459,-64.810,170.686,28.244,155.338
C00642=1055.879,-99.709,-64.801,170.684,28.243,155.338
C00643=1055.872,-99.958,-64.791,170.682,28.242,155.338
C00644=1055.866,-100.208,-64.779,170.680,28.242,155.338
C00645=1055.860,-100.458,-64.770,170.679,28.240,155.338
C00646=1055.854,-100.708,-64.760,170.676,28.239,155.338
C00647=1055.848,-100.957,-64.749,170.674,28.238,155.338
C00648=1055.842,-101.207,-64.740,170.672,28.238,155.338
C00649=1055.835,-101.456,-64.729,170.670,28.237,155.338
C00650=1055.830,-101.706,-64.719,170.668,28.236,155.338
C00651=1055.823,-101.956,-64.709,170.667,28.235,155.338
C00652=1055.817,-102.206,-64.699,170.665,28.234,155.338
C00653=1055.811,-102.456,-64.688,170.663,28.233,155.338
C00654=1055.805,-102.705,-64.679,170.660,28.232,155.338
C00655=1055.798,-102.955,-64.668,170.658,28.231,155.338
C00656=1055.793,-103.205,-64.658,170.656,28.230,155.338
C00657=1055.787,-103.455,-64.649,170.655,28.230,155.338
C00658=1055.780,-103.704,-64.638,170.653,28.229,155.338
C00659=1055.773,-103.954,-64.628,170.651,28.228,155.338
C00660=1055.768,-104.204,-64.617,170.649,28.227,155.339
C00661=1055.762,-104.453,-64.608,170.647,28.226,155.338
C00662=1055.755,-104.703,-64.598,170.644,28.225,155.338
C00663=1055.750,-104.953,-64.587,170.642,28.224,155.339
C00664=1055.743,-105.203,-64.578,170.641,28.223,155.339
C00665=1055.737,-105.452,-64.568,170.639,28.223,155.339
C00666=1055.731,-105.702,-64.558,170.637,28.222,155.339
C00667=1055.725,-105.952,-64.548,170.635,28.221,155.339
C00668=1055.719,-106.201,-64.538,170.633,28.220,155.339
C00669=1055.713,-106.451,-64.528,170.631,28.219,155.339
C00670=1055.707,-106.700,-64.518,170.629,28.218,155.339
C00671=1055.701,-106.951,-64.508,170.627,28.217,155.339
C00672=1055.695,-107.200,-64.498,170.625,28.217,155.339
C00673=1055.688,-107.450,-64.488,170.623,28.216,155.339
C00674=1055.682,-107.700,-64.479,170.621,28.215,155.339
C00675=1055.676,-107.950,-64.469,170.619,28.214,155.339
C00676=1055.670,-108.199,-64.458,170.617,28.214,155.339
C00677=1055.664,-108.449,-64.449,170.615,28.213,155.339
C00678=1055.657,-108.699,-64.439,170.613,28.212,155.339
C00679=1055.651,-108.949,-64.429,170.611,28.211,155.339
C00680=1055.645,-109.198,-64.419,170.609,28.211,155.339
C00681=1055.639,-109.448,-64.410,170.607,28.210,155.339
C00682=1055.632,-109.697,-64.400,170.605,28.209,155.339
C00683=1055.626,-109.947,-64.390,170.603,28.209,155.339
C00684=1055.621,-110.197,-64.380,170.602,28.208,155.339
C00685=1055.614,-110.447,-64.370,170.599,28.207,155.339
C00686=1055.608,-110.696,-64.360,170.597,28.206,155.339
C00687=1055.602,-110.946,-64.351,170.595,28.205,155.339
C00688=1055.596,-111.196,-64.341,170.593,28.205,155.339
C00689=1055.590,-111.446,-64.332,170.591,28.204,155.339
C00690=1055.583,-111.696,-64.322,170.589,28.203,155.340
C00691=1055.577,-111.945,-64.312,170.587,28.202,155.340
C00692=1055.571,-112.195,-64.302,170.585,28.202,155.340
C00693=1055.565,-112.444,-64.293,170.583,28.201,155.340
C00694=1055.558,-112.694,-64.283,170.581,28.200,155.340
C00695=1055.553,-112.944,-64.273,170.579,28.200,155.340
C00696=1055.547,-113.194,-64.263,170.577,28.199,155.340
C00697=1055.541,-113.444,-64.254,170.575,28.198,155.340
C00698=1055.535,-113.694,-64.244,170.573,28.198,155.340
C00699=1055.528,-113.943,-64.235,170.571,28.197,155.340
C00700=1055.522,-114.193,-64.225,170.569,28.196,155.340
C00701=1055.516,-114.442,-64.215,170.567,28.195,155.340
C00702=1055.509,-114.727,-64.205,170.565,28.195,155.340
C00703=1055.502,-115.010,-64.194,170.562,28.194,155.340
C00704=1055.495,-115.295,-64.182,170.560,28.193,155.340
C00705=1055.488,-115.579,-64.172,170.558,28.193,155.340
C00706=1055.482,-115.829,-64.162,170.555,28.192,155.341
C00707=1055.476,-116.078,-64.153,170.554,28.191,155.341
C00708=1055.470,-116.328,-64.143,170.552,28.191,155.341
C00709=1055.464,-116.578,-64.134,170.550,28.190,155.341
C00710=1055.457,-116.828,-64.124,170.548,28.190,155.341
C00711=1055.452,-117.077,-64.115,170.546,28.189,155.341
C00712=1055.446,-117.327,-64.105,170.544,28.188,155.341
C00713=1055.440,-117.576,-64.096,170.541,28.187,155.341
C00714=1055.433,-117.826,-64.087,170.539,28.187,155.341
C00715=1055.426,-118.076,-64.077,170.538,28.186,155.341
C00716=1055.420,-118.326,-64.068,170.536,28.186,155.341
C00717=1055.414,-118.575,-64.058,170.534,28.185,155.341
C00718=1055.408,-118.825,-64.049,170.532,28.184,155.341
C00719=1055.402,-119.075,-64.039,170.530,28.184,155.341
C00720=1055.396,-119.325,-64.030,170.527,28.183,155.342
C00721=1055.390,-119.574,-64.020,170.525,28.183,155.342
C00722=1055.384,-119.824,-64.011,170.523,28.182,155.342
C00723=1055.378,-120.074,-64.002,170.521,28.182,155.342
C00724=1055.371,-120.324,-63.993,170.520,28.181,155.342
C00725=1055.365,-120.573,-63.983,170.518,28.180,155.342
C00726=1055.359,-120.823,-63.974,170.516,28.180,155.342
C00727=1055.353,-121.073,-63.964,170.513,28.179,155.342
C00728=1055.347,-121.322,-63.955,170.511,28.179,155.342
C00729=1055.341,-121.572,-63.945,170.509,28.178,155.342
C00730=1055.335,-121.822,-63.937,170.507,28.178,155.342
C00731=1055.329,-122.072,-63.927,170.505,28.177,155.342
C00732=1055.322,-122.322,-63.918,170.503,28.177,155.342
C00733=1055.316,-122.571,-63.908,170.502,28.177,155.343
C00734=1055.310,-122.820,-63.899,170.499,28.176,155.343
C00735=1055.304,-123.071,-63.890,170.497,28.175,155.343
C00736=1055.298,-123.321,-63.881,170.495,28.175,155.343
C00737=1055.292,-123.570,-63.871,170.493,28.174,155.343
C00738=1055.285,-123.820,-63.862,170.491,28.174,155.343
C00739=1055.279,-124.070,-63.853,170.489,28.174,155.343
C00740=1055.274,-124.319,-63.844,170.487,28.173,155.343
C00741=1055.267,-124.569,-63.835,170.485,28.173,155.343
C00742=1055.261,-124.819,-63.825,170.483,28.172,155.343
C00743=1055.255,-125.069,-63.817,170.481,28.171,155.344
C00744=1055.248,-125.319,-63.807,170.479,28.171,155.344
C00745=1055.243,-125.568,-63.798,170.477,28.171,155.344
C00746=1055.236,-125.818,-63.789,170.475,28.170,155.344
C00747=1055.230,-126.068,-63.780,170.473,28.170,155.344
C00748=1055.224,-126.318,-63.771,170.470,28.170,155.344
C00749=1055.218,-126.568,-63.761,170.468,28.169,155.344
C00750=1055.212,-126.817,-63.753,170.466,28.169,155.344
C00751=1055.206,-127.067,-63.744,170.464,28.168,155.344
C00752=1055.199,-127.317,-63.734,170.462,28.168,155.344
C00753=1055.193,-127.567,-63.726,170.461,28.167,155.345
C00754=1055.187,-127.816,-63.717,170.459,28.167,155.345
C00755=1055.182,-128.066,-63.707,170.457,28.166,155.345
C00756=1055.178,-128.316,-63.697,170.455,28.165,155.345
C00757=1055.175,-128.566,-63.686,170.453,28.163,155.344
C00758=1055.174,-128.817,-63.675,170.452,28.161,155.344
C00759=1055.174,-129.067,-63.662,170.450,28.157,155.344
C00760=1055.174,-129.318,-63.649,170.449,28.154,155.343
C00761=1055.176,-129.567,-63.636,170.448,28.150,155.343
C00762=1055.179,-129.819,-63.621,170.447,28.145,155.342
C00763=1055.184,-130.070,-63.606,170.447,28.140,155.341
C00764=1055.190,-130.321,-63.590,170.445,28.135,155.340
C00765=1055.196,-130.571,-63.573,170.445,28.128,155.339
C00766=1054.825,-130.594,-63.784,170.397,28.295,155.372
C00767=1054.818,-130.344,-63.800,170.399,28.301,155.373
C00768=1054.813,-130.093,-63.816,170.399,28.307,155.374
C00769=1054.808,-129.843,-63.831,170.399,28.312,155.375
C00770=1054.804,-129.591,-63.845,170.400,28.316,155.376
C00771=1054.802,-129.341,-63.859,170.401,28.320,155.376
C00772=1054.801,-129.091,-63.872,170.402,28.324,155.377
C00773=1054.802,-128.840,-63.884,170.404,28.327,155.377
C00774=1054.804,-128.590,-63.896,170.405,28.329,155.378
C00775=1054.806,-128.339,-63.907,170.407,28.331,155.378
C00776=1054.810,-128.089,-63.917,170.409,28.333,155.378
C00777=1054.815,-127.840,-63.927,170.411,28.333,155.378
C00778=1054.821,-127.589,-63.936,170.413,28.334,155.378
C00779=1054.828,-127.340,-63.945,170.415,28.334,155.378
C00780=1054.833,-127.091,-63.954,170.417,28.335,155.378
C00781=1054.839,-126.840,-63.963,170.419,28.335,155.377
C00782=1054.846,-126.591,-63.972,170.421,28.336,155.377
C00783=1054.852,-126.341,-63.982,170.423,28.336,155.377
C00784=1054.858,-126.091,-63.990,170.425,28.336,155.377
C00785=1054.863,-125.841,-64.000,170.427,28.336,155.377
C00786=1054.870,-125.592,-64.009,170.429,28.337,155.377
C00787=1054.876,-125.342,-64.017,170.431,28.337,155.377
C00788=1054.882,-125.092,-64.027,170.433,28.338,155.377
C00789=1054.889,-124.842,-64.036,170.436,28.338,155.377
C00790=1054.895,-124.593,-64.045,170.438,28.339,155.376
C00791=1054.901,-124.343,-64.054,170.440,28.339,155.376
C00792=1054.907,-124.093,-64.064,170.441,28.340,155.376
C00793=1054.913,-123.843,-64.073,170.443,28.340,155.376
C00794=1054.920,-123.593,-64.081,170.445,28.341,155.376
C00795=1054.925,-123.344,-64.091,170.447,28.341,155.376
C00796=1054.931,-123.094,-64.100,170.450,28.342,155.376
C00797=1054.938,-122.844,-64.110,170.452,28.342,155.376
C00798=1054.944,-122.595,-64.119,170.454,28.343,155.376
C00799=1054.950,-122.344,-64.128,170.456,28.343,155.376
C00800=1054.957,-122.095,-64.137,170.458,28.344,155.376
C00801=1054.962,-121.846,-64.146,170.460,28.344,155.376
C00802=1054.968,-121.596,-64.156,170.462,28.345,155.375
C00803=1054.974,-121.346,-64.166,170.464,28.345,155.375
C00804=1054.981,-121.096,-64.175,170.466,28.346,155.375
C00805=1054.987,-120.846,-64.184,170.468,28.346,155.375
C00806=1054.993,-120.596,-64.194,170.470,28.347,155.375
C00807=1054.998,-120.347,-64.203,170.472,28.347,155.375
C00808=1055.005,-120.097,-64.212,170.474,28.347,155.375
C00809=1055.011,-119.848,-64.221,170.477,28.348,155.375
C00810=1055.018,-119.598,-64.231,170.479,28.349,155.375
C00811=1055.024,-119.348,-64.240,170.480,28.350,155.375
C00812=1055.030,-119.098,-64.249,170.482,28.350,155.375
C00813=1055.036,-118.848,-64.259,170.484,28.351,155.374
C00814=1055.042,-118.598,-64.268,170.486,28.351,155.374
C00815=1055.047,-118.349,-64.278,170.488,28.351,155.374
C00816=1055.054,-118.099,-64.287,170.491,28.352,155.374
C00817=1055.060,-117.849,-64.297,170.493,28.353,155.374
C00818=1055.067,-117.600,-64.306,170.495,28.354,155.374
C00819=1055.073,-117.350,-64.315,170.497,28.354,155.374
C00820=1055.079,-117.100,-64.325,170.498,28.355,155.374
C00821=1055.085,-116.850,-64.334,170.500,28.355,155.374
C00822=1055.091,-116.601,-64.344,170.502,28.355,155.374
C00823=1055.098,-116.351,-64.354,170.505,28.357,155.374
C00824=1055.104,-116.101,-64.363,170.507,28.357,155.374
C00825=1055.110,-115.851,-64.373,170.509,28.358,155.374
C00826=1055.116,-115.601,-64.382,170.511,28.358,155.374
C00827=1055.123,-115.318,-64.393,170.513,28.359,155.373
C00828=1055.130,-115.034,-64.403,170.515,28.360,155.373
C00829=1055.137,-114.749,-64.415,170.517,28.360,155.373
C00830=1055.144,-114.466,-64.426,170.520,28.361,155.373
C00831=1055.150,-114.216,-64.435,170.522,28.362,155.373
C00832=1055.156,-113.966,-64.445,170.524,28.362,155.373
C00833=1055.162,-113.716,-64.454,170.526,28.363,155.373
C00834=1055.169,-113.466,-64.464,170.528,28.364,155.373
C00835=1055.175,-113.217,-64.474,170.530,28.364,155.373
C00836=1055.180,-112.966,-64.484,170.532,28.365,155.373
C00837=1055.186,-112.717,-64.493,170.534,28.366,155.373
C00838=1055.192,-112.467,-64.503,170.536,28.367,155.373
C00839=1055.199,-112.217,-64.512,170.538,28.367,155.373
C00840=1055.205,-111.968,-64.523,170.540,28.368,155.373
C00841=1055.211,-111.718,-64.532,170.542,28.369,155.373
C00842=1055.217,-111.468,-64.542,170.544,28.369,155.373
C00843=1055.224,-111.219,-64.551,170.547,28.370,155.373
C00844=1055.230,-110.969,-64.561,170.548,28.371,155.373
C00845=1055.236,-110.719,-64.571,170.550,28.372,155.373
C00846=1055.242,-110.470,-64.581,170.552,28.372,155.372
C00847=1055.248,-110.220,-64.591,170.554,28.373,155.372
C00848=1055.254,-109.970,-64.601,170.556,28.374,155.372
C00849=1055.260,-109.720,-64.610,170.558,28.374,155.372
C00850=1055.266,-109.470,-64.620,170.561,28.375,155.372
C00851=1055.273,-109.221,-64.630,170.562,28.376,155.372
C00852=1055.279,-108.971,-64.640,170.564,28.376,155.372
C00853=1055.285,-108.721,-64.649,170.566,28.377,155.372
C00854=1055.291,-108.472,-64.659,170.568,28.378,155.372
C00855=1055.297,-108.222,-64.669,170.570,28.379,155.372
C00856=1055.303,-107.972,-64.679,170.572,28.379,155.372
C00857=1055.309,-107.723,-64.689,170.575,28.381,155.372
C00858=1055.316,-107.473,-64.698,170.577,28.381,155.372
C00859=1055.322,-107.224,-64.709,170.578,28.382,155.372
C00860=1055.328,-106.974,-64.718,170.580,28.383,155.372
C00861=1055.334,-106.724,-64.728,170.582,28.384,155.372
C00862=1055.340,-106.474,-64.738,170.584,28.384,155.372
C00863=1055.346,-106.225,-64.748,170.586,28.385,155.372
C00864=1055.353,-105.975,-64.758,170.589,28.386,155.372
C00865=1055.359,-105.724,-64.768,170.591,28.387,155.372
C00866=1055.365,-105.475,-64.779,170.592,28.388,155.372
C00867=1055.371,-105.225,-64.788,170.594,28.388,155.372
C00868=1055.377,-104.975,-64.798,170.596,28.389,155.372
C00869=1055.383,-104.726,-64.809,170.598,28.390,155.372
C00870=1055.389,-104.476,-64.818,170.600,28.391,155.372
C00871=1055.396,-104.227,-64.828,170.602,28.392,155.372
C00872=1055.401,-103.977,-64.839,170.605,28.393,155.372
C00873=1055.407,-103.727,-64.848,170.606,28.394,155.372
C00874=1055.414,-103.478,-64.858,170.608,28.394,155.371
C00875=1055.419,-103.228,-64.869,170.610,28.395,155.372
C00876=1055.426,-102.978,-64.879,170.612,28.396,155.372
C00877=1055.433,-102.728,-64.889,170.614,28.397,155.371
C00878=1055.439,-102.478,-64.898,170.616,28.398,155.371
C00879=1055.444,-102.229,-64.909,170.617,28.399,155.372
C00880=1055.451,-101.979,-64.919,170.620,28.400,155.371
C00881=1055.457,-101.730,-64.929,170.622,28.401,155.371
C00882=1055.463,-101.480,-64.939,170.624,28.402,155.371
C00883=1055.469,-101.230,-64.949,170.626,28.402,155.371
C00884=1055.476,-100.980,-64.959,170.628,28.403,155.371
C00885=1055.482,-100.730,-64.970,170.630,28.404,155.371
C00886=1055.488,-100.481,-64.980,170.631,28.405,155.371
C00887=1055.494,-100.232,-64.990,170.633,28.406,155.371
C00888=1055.500,-99.981,-65.000,170.636,28.407,155.371
C00889=1055.506,-99.732,-65.011,170.638,28.408,155.371
C00890=1055.512,-99.481,-65.021,170.640,28.409,155.371
C00891=1055.520,-99.197,-65.032,170.642,28.410,155.371
C00892=1055.527,-98.911,-65.044,170.644,28.411,155.371
C00893=1055.534,-98.625,-65.056,170.646,28.412,155.371
C00894=1055.541,-98.340,-65.068,170.649,28.413,155.371
C00895=1055.547,-98.090,-65.078,170.651,28.414,155.371
C00896=1055.553,-97.840,-65.088,170.653,28.415,155.371
C00897=1055.559,-97.591,-65.098,170.655,28.416,155.371
C00898=1055.565,-97.340,-65.109,170.656,28.417,155.371
C00899=1055.572,-97.091,-65.119,170.658,28.418,155.371
C00900=1055.577,-96.841,-65.130,170.660,28.419,155.371
C00901=1055.584,-96.592,-65.140,170.662,28.420,155.371
C00902=1055.590,-96.343,-65.151,170.665,28.421,155.371
C00903=1055.595,-96.092,-65.161,170.666,28.422,155.371
C00904=1055.602,-95.843,-65.172,170.668,28.423,155.371
C00905=1055.608,-95.593,-65.182,170.670,28.424,155.372
C00906=1055.614,-95.343,-65.192,170.672,28.425,155.372
C00907=1055.620,-95.094,-65.203,170.674,28.426,155.371
C00908=1055.625,-94.844,-65.214,170.676,28.427,155.371
C00909=1055.632,-94.594,-65.224,170.677,28.428,155.372
C00910=1055.638,-94.344,-65.235,170.679,28.429,155.372
C00911=1055.644,-94.095,-65.245,170.682,28.430,155.372
C00912=1055.650,-93.845,-65.255,170.684,28.431,155.372
C00913=1055.656,-93.595,-65.266,170.686,28.432,155.372
C00914=1055.663,-93.346,-65.277,170.688,28.433,155.372
C00915=1055.668,-93.096,-65.287,170.689,28.435,155.372
C00916=1055.675,-92.846,-65.297,170.691,28.436,155.372
C00917=1055.680,-92.597,-65.308,170.693,28.437,155.372
C00918=1055.687,-92.347,-65.319,170.695,28.438,155.372
C00919=1055.693,-92.097,-65.329,170.698,28.439,155.372
C00920=1055.699,-91.847,-65.340,170.699,28.440,155.372
C00921=1055.706,-91.597,-65.350,170.701,28.441,155.372
C00922=1055.711,-91.348,-65.361,170.703,28.442,155.372
C00923=1055.717,-91.099,-65.372,170.705,28.443,155.372
C00924=1055.724,-90.849,-65.382,170.707,28.445,155.372
C00925=1055.730,-90.599,-65.393,170.709,28.446,155.372
C00926=1055.735,-90.349,-65.404,170.710,28.447,155.372
C00927=1055.742,-90.100,-65.414,170.712,28.448,155.372
C00928=1055.748,-89.850,-65.425,170.715,28.449,155.372
C00929=1055.754,-89.600,-65.436,170.717,28.450,155.372
C00930=1055.760,-89.351,-65.446,170.719,28.451,155.372
C00931=1055.767,-89.101,-65.458,170.720,28.452,155.372
C00932=1055.772,-88.851,-65.468,170.722,28.453,155.372
C00933=1055.779,-88.602,-65.478,170.724,28.454,155.372
C00934=1055.785,-88.351,-65.489,170.726,28.456,155.372
C00935=1055.791,-88.102,-65.500,170.728,28.457,155.372
C00936=1055.797,-87.853,-65.510,170.730,28.458,155.372
C00937=1055.804,-87.602,-65.522,170.731,28.459,155.372
C00938=1055.809,-87.353,-65.533,170.734,28.461,155.372
C00939=1055.816,-87.104,-65.543,170.736,28.462,155.373
C00940=1055.822,-86.854,-65.554,170.738,28.463,155.373
C00941=1055.828,-86.604,-65.565,170.740,28.464,155.373
C00942=1055.834,-86.355,-65.575,170.741,28.465,155.373
C00943=1055.841,-86.105,-65.587,170.743,28.466,155.373
C00944=1055.846,-85.855,-65.597,170.745,28.467,155.373
C00945=1055.853,-85.605,-65.607,170.747,28.469,155.373
C00946=1055.859,-85.355,-65.618,170.749,28.470,155.373
C00947=1055.865,-85.106,-65.629,170.751,28.471,155.373
C00948=1055.872,-84.856,-65.640,170.753,28.472,155.373
C00949=1055.878,-84.606,-65.651,170.755,28.473,155.373
C00950=1055.884,-84.356,-65.662,170.757,28.474,155.373
C00951=1055.890,-84.107,-65.672,170.759,28.476,155.373
C00952=1055.896,-83.858,-65.684,170.761,28.477,155.373
C00953=1055.903,-83.608,-65.695,170.762,28.478,155.373
C00954=1055.908,-83.358,-65.706,170.764,28.479,155.373
C00955=1055.916,-83.075,-65.718,170.767,28.480,155.373
C00956=1055.923,-82.791,-65.730,170.769,28.482,155.373
C00957=1055.930,-82.508,-65.742,170.771,28.483,155.373
C00958=1055.937,-82.225,-65.755,170.773,28.485,155.373
C00959=1055.943,-81.976,-65.766,170.775,28.486,155.373
C00960=1055.950,-81.726,-65.777,170.777,28.487,155.373
C00961=1055.956,-81.476,-65.788,170.779,28.488,155.374
C00962=1055.962,-81.226,-65.799,170.781,28.489,155.374
C00963=1055.968,-80.977,-65.810,170.782,28.491,155.374
C00964=1055.975,-80.727,-65.820,170.784,28.492,155.374
C00965=1055.981,-80.478,-65.832,170.787,28.493,155.374
C00966=1055.987,-80.228,-65.843,170.789,28.494,155.374
C00967=1055.993,-79.978,-65.854,170.790,28.496,155.374
C00968=1056.000,-79.728,-65.865,170.792,28.497,155.374
C00969=1056.006,-79.479,-65.876,170.794,28.498,155.374
C00970=1056.012,-79.229,-65.887,170.796,28.499,155.374
C00971=1056.018,-78.980,-65.898,170.798,28.500,155.374
C00972=1056.025,-78.730,-65.910,170.799,28.502,155.374
C00973=1056.030,-78.480,-65.921,170.801,28.503,155.374
C00974=1056.037,-78.230,-65.932,170.803,28.504,155.374
C00975=1056.042,-77.980,-65.943,170.805,28.506,155.374
C00976=1056.049,-77.731,-65.955,170.808,28.507,155.374
C00977=1056.055,-77.481,-65.966,170.809,28.509,155.375
C00978=1056.061,-77.231,-65.977,170.811,28.510,155.375
C00979=1056.067,-76.982,-65.988,170.813,28.511,155.375
C00980=1056.073,-76.732,-66.000,170.815,28.512,155.375
C00981=1056.079,-76.483,-66.011,170.817,28.513,155.375
C00982=1056.086,-76.232,-66.022,170.818,28.515,155.375
C00983=1056.092,-75.983,-66.033,170.820,28.516,155.375
C00984=1056.098,-75.733,-66.045,170.822,28.518,155.375
C00985=1056.104,-75.484,-66.055,170.824,28.519,155.375
C00986=1056.110,-75.234,-66.067,170.826,28.520,155.375
C00987=1056.116,-74.985,-66.078,170.827,28.522,155.375
C00988=1056.122,-74.735,-66.090,170.830,28.523,155.376
C00989=1056.128,-74.485,-66.100,170.832,28.524,155.376
C00990=1056.135,-74.235,-66.112,170.834,28.526,155.376
C00991=1056.141,-73.986,-66.123,170.836,28.527,155.376
C00992=1056.147,-73.736,-66.135,170.837,28.529,155.376
C00993=1056.153,-73.487,-66.146,170.839,28.530,155.376
C00994=1056.159,-73.237,-66.157,170.841,28.531,155.376
C00995=1056.166,-72.987,-66.169,170.843,28.533,155.376
C00996=1056.171,-72.737,-66.181,170.844,28.534,155.376
C00997=1056.177,-72.487,-66.192,170.846,28.536,155.376
C00998=1056.183,-72.238,-66.204,170.848,28.537,155.377
C00999=1056.190,-71.988,-66.215,170.850,28.539,155.377
C01000=1056.196,-71.739,-66.226,170.852,28.540,155.377
C01001=1056.201,-71.489,-66.238,170.853,28.542,155.377
C01002=1056.207,-71.240,-66.250,170.856,28.543,155.377
C01003=1056.214,-70.990,-66.261,170.858,28.545,155.377
C01004=1056.220,-70.741,-66.273,170.860,28.546,155.377
C01005=1056.225,-70.490,-66.285,170.861,28.548,155.377
C01006=1056.231,-70.241,-66.296,170.863,28.549,155.377
C01007=1056.238,-69.991,-66.307,170.865,28.551,155.377
C01008=1056.244,-69.742,-66.319,170.867,28.552,155.378
C01009=1056.249,-69.492,-66.331,170.868,28.553,155.378
C01010=1056.256,-69.242,-66.343,170.870,28.555,155.378
C01011=1056.262,-68.993,-66.354,170.872,28.557,155.378
C01012=1056.268,-68.743,-66.366,170.874,28.558,155.378
C01013=1056.273,-68.493,-66.377,170.876,28.559,155.378
C01014=1056.280,-68.244,-66.389,170.877,28.561,155.378
C01015=1056.286,-67.994,-66.400,170.879,28.563,155.378
C01016=1056.292,-67.745,-66.412,170.881,28.564,155.379
C01017=1056.298,-67.495,-66.424,170.883,28.565,155.379
C01018=1056.305,-67.245,-66.436,170.885,28.567,155.379
C01019=1056.312,-66.964,-66.448,170.887,28.569,155.379
C01020=1056.318,-66.682,-66.462,170.889,28.571,155.379
C01021=1056.326,-66.402,-66.475,170.891,28.572,155.379
C01022=1056.332,-66.121,-66.489,170.893,28.574,155.379
C01023=1056.338,-65.871,-66.499,170.895,28.576,155.379
C01024=1056.345,-65.622,-66.511,170.897,28.577,155.380
C01025=1056.351,-65.372,-66.524,170.899,28.578,155.380
C01026=1056.356,-65.122,-66.535,170.900,28.580,155.380
C01027=1056.363,-64.873,-66.547,170.902,28.582,155.380
C01028=1056.369,-64.623,-66.559,170.904,28.583,155.380
C01029=1056.375,-64.373,-66.570,170.906,28.584,155.380
C01030=1056.381,-64.124,-66.582,170.908,28.586,155.380
C01031=1056.387,-63.874,-66.595,170.909,28.588,155.380
C01032=1056.393,-63.624,-66.606,170.911,28.589,155.381
C01033=1056.400,-63.375,-66.618,170.913,28.591,155.381
C01034=1056.406,-63.125,-66.630,170.915,28.593,155.381
C01035=1056.411,-62.876,-66.642,170.917,28.594,155.381
C01036=1056.418,-62.626,-66.653,170.919,28.595,155.381
C01037=1056.424,-62.376,-66.665,170.921,28.597,155.381
C01038=1056.430,-62.126,-66.678,170.923,28.599,155.381
C01039=1056.436,-61.877,-66.689,170.924,28.600,155.381
C01040=1056.443,-61.627,-66.700,170.926,28.602,155.382
C01041=1056.449,-61.377,-66.713,170.928,28.603,155.382
C01042=1056.455,-61.128,-66.725,170.930,28.605,155.382
C01043=1056.461,-60.879,-66.736,170.931,28.606,155.382
C01044=1056.467,-60.628,-66.748,170.933,28.608,155.382
C01045=1056.474,-60.379,-66.760,170.935,28.610,155.382
C01046=1056.480,-60.129,-66.772,170.937,28.611,155.382
C01047=1056.486,-59.880,-66.784,170.938,28.613,155.382
C01048=1056.492,-59.631,-66.796,170.940,28.614,155.382
C01049=1056.499,-59.381,-66.808,170.942,28.616,155.383
C01050=1056.504,-59.130,-66.820,170.944,28.617,155.383
C01051=1056.511,-58.882,-66.832,170.946,28.619,155.383
C01052=1056.516,-58.632,-66.844,170.947,28.621,155.383
C01053=1056.523,-58.382,-66.856,170.949,28.622,155.383
C01054=1056.530,-58.133,-66.868,170.951,28.624,155.383
C01055=1056.536,-57.883,-66.881,170.953,28.625,155.384
C01056=1056.542,-57.633,-66.893,170.954,28.627,155.384
C01057=1056.548,-57.384,-66.904,170.957,28.628,155.384
C01058=1056.554,-57.134,-66.916,170.959,28.630,155.384
C01059=1056.561,-56.884,-66.928,170.961,28.632,155.384
C01060=1056.567,-56.635,-66.940,170.962,28.633,155.384
C01061=1056.573,-56.385,-66.953,170.964,28.635,155.384
C01062=1056.580,-56.135,-66.965,170.966,28.637,155.384
C01063=1056.585,-55.886,-66.977,170.968,28.638,155.385
C01064=1056.592,-55.636,-66.989,170.969,28.640,155.385
C01065=1056.598,-55.387,-67.001,170.971,28.642,155.385
C01066=1056.604,-55.137,-67.013,170.973,28.643,155.385
C01067=1056.611,-54.887,-67.025,170.975,28.645,155.385
C01068=1056.617,-54.637,-67.038,170.976,28.646,155.385
C01069=1056.623,-54.388,-67.050,170.978,28.648,155.385
C01070=1056.630,-54.138,-67.062,170.980,28.650,155.386
C01071=1056.635,-53.889,-67.074,170.982,28.651,155.386
C01072=1056.642,-53.640,-67.086,170.983,28.653,155.386
C01073=1056.648,-53.390,-67.098,170.985,28.655,155.386
C01074=1056.655,-53.140,-67.110,170.987,28.656,155.386
C01075=1056.661,-52.891,-67.122,170.989,28.657,155.386
C01076=1056.667,-52.641,-67.135,170.991,28.659,155.386
C01077=1056.674,-52.391,-67.147,170.992,28.661,155.387
C01078=1056.680,-52.141,-67.159,170.994,28.662,155.387
C01079=1056.686,-51.892,-67.171,170.996,28.664,155.387
C01080=1056.692,-51.642,-67.184,170.998,28.665,155.387
C01081=1056.699,-51.392,-67.196,170.999,28.667,155.387
C01082=1056.706,-51.143,-67.208,171.001,28.669,155.387
C01083=1056.712,-50.863,-67.222,171.004,28.671,155.388
C01084=1056.719,-50.584,-67.235,171.006,28.673,155.388
C01085=1056.727,-50.304,-67.250,171.007,28.674,155.388
C01086=1056.733,-50.024,-67.263,171.009,28.677,155.388
C01087=1056.739,-49.774,-67.276,171.011,28.678,155.388
C01088=1056.746,-49.525,-67.288,171.012,28.680,155.388
C01089=1056.752,-49.275,-67.301,171.014,28.682,155.389
C01090=1056.758,-49.025,-67.314,171.017,28.683,155.389
C01091=1056.763,-48.775,-67.326,171.019,28.686,155.389
C01092=1056.770,-48.526,-67.338,171.020,28.687,155.389
C01093=1056.776,-48.277,-67.351,171.022,28.689,155.389
C01094=1056.782,-48.027,-67.364,171.024,28.691,155.389
C01095=1056.788,-47.777,-67.376,171.026,28.693,155.390
C01096=1056.794,-47.528,-67.388,171.027,28.695,155.390
C01097=1056.800,-47.278,-67.401,171.029,28.696,155.390
C01098=1056.806,-47.029,-67.414,171.031,28.698,155.390
C01099=1056.813,-46.779,-67.426,171.033,28.700,155.390
C01100=1056.819,-46.529,-67.438,171.034,28.702,155.390
C01101=1056.825,-46.279,-67.451,171.036,28.703,155.391
C01102=1056.831,-46.030,-67.464,171.038,28.705,155.391
C01103=1056.837,-45.780,-67.477,171.040,28.707,155.391
C01104=1056.844,-45.531,-67.489,171.041,28.709,155.391
C01105=1056.850,-45.281,-67.502,171.043,28.710,155.391
C01106=1056.856,-45.031,-67.515,171.045,28.712,155.392
C01107=1056.862,-44.782,-67.527,171.047,28.714,155.392
C01108=1056.869,-44.533,-67.540,171.048,28.716,155.392
C01109=1056.874,-44.283,-67.552,171.050,28.718,155.392
C01110=1056.880,-44.033,-67.565,171.052,28.720,155.392
C01111=1056.887,-43.784,-67.578,171.053,28.721,155.392
C01112=1056.892,-43.534,-67.591,171.055,28.723,155.393
C01113=1056.899,-43.284,-67.603,171.057,28.725,155.393
C01114=1056.905,-43.035,-67.616,171.059,28.727,155.393
C01115=1056.911,-42.785,-67.628,171.060,28.729,155.393
C01116=1056.917,-42.535,-67.641,171.062,28.730,155.393
C01117=1056.924,-42.286,-67.654,171.064,28.732,155.394
C01118=1056.930,-42.036,-67.666,171.066,28.734,155.394
C01119=1056.936,-41.787,-67.680,171.067,28.736,155.394
C01120=1056.942,-41.537,-67.692,171.069,28.737,155.394
C01121=1056.948,-41.287,-67.705,171.071,28.740,155.394
C01122=1056.954,-41.038,-67.718,171.072,28.741,155.395
C01123=1056.961,-40.788,-67.730,171.073,28.743,155.395
C01124=1056.967,-40.539,-67.743,171.075,28.745,155.395
C01125=1056.973,-40.289,-67.756,171.077,28.746,155.395
C01126=1056.979,-40.040,-67.769,171.079,28.748,155.395
C01127=1056.985,-39.790,-67.781,171.080,28.750,155.396
C01128=1056.992,-39.541,-67.794,171.082,28.752,155.396
C01129=1056.998,-39.291,-67.807,171.084,28.754,155.396
C01130=1057.005,-39.041,-67.820,171.086,28.756,155.396
C01131=1057.011,-38.791,-67.833,171.087,28.757,155.396
C01132=1057.017,-38.542,-67.846,171.089,28.760,155.397
C01133=1057.023,-38.292,-67.859,171.091,28.761,155.397
C01134=1057.029,-38.043,-67.872,171.093,28.763,155.397
C01135=1057.035,-37.793,-67.885,171.094,28.765,155.397
C01136=1057.041,-37.544,-67.898,171.096,28.767,155.397
C01137=1057.047,-37.294,-67.910,171.098,28.769,155.398
C01138=1057.053,-37.045,-67.924,171.099,28.771,155.398
C01139=1057.059,-36.795,-67.936,171.101,28.773,155.398
C01140=1057.065,-36.546,-67.949,171.103,28.774,155.398
C01141=1057.072,-36.296,-67.963,171.105,28.777,155.398
C01142=1057.078,-36.046,-67.975,171.106,28.778,155.398
C01143=1057.084,-35.796,-67.989,171.108,28.781,155.399
C01144=1057.090,-35.547,-68.001,171.110,28.782,155.399
C01145=1057.097,-35.297,-68.015,171.111,28.784,155.399
C01146=1057.103,-35.048,-68.028,171.113,28.786,155.399
C01147=1057.109,-34.769,-68.042,171.115,28.788,155.400
C01148=1057.116,-34.489,-68.057,171.117,28.791,155.400
C01149=1057.123,-34.210,-68.072,171.119,28.793,155.400
C01150=1057.130,-33.931,-68.087,171.121,28.795,155.400
C01151=1057.136,-33.681,-68.100,171.123,28.797,155.401
C01152=1057.142,-33.431,-68.113,171.124,28.799,155.401
C01153=1057.148,-33.181,-68.126,171.126,28.801,155.401
C01154=1057.155,-32.932,-68.139,171.128,28.803,155.401
C01155=1057.161,-32.682,-68.152,171.130,28.805,155.401
C01156=1057.167,-32.433,-68.165,171.131,28.807,155.402
C01157=1057.173,-32.184,-68.179,171.133,28.808,155.402
C01158=1057.179,-31.934,-68.192,171.134,28.810,155.402
C01159=1057.186,-31.684,-68.205,171.136,28.813,155.402
C01160=1057.191,-31.434,-68.219,171.137,28.814,155.402
C01161=1057.197,-31.185,-68.232,171.139,28.816,155.403
C01162=1057.204,-30.936,-68.245,171.141,28.818,155.403
C01163=1057.210,-30.686,-68.258,171.142,28.820,155.403
C01164=1057.216,-30.437,-68.271,171.144,28.822,155.403
C01165=1057.223,-30.187,-68.285,171.146,28.824,155.404
C01166=1057.229,-29.937,-68.298,171.148,28.826,155.404
C01167=1057.235,-29.688,-68.311,171.149,28.828,155.404
C01168=1057.241,-29.438,-68.324,171.151,28.830,155.404
C01169=1057.248,-29.188,-68.337,171.153,28.832,155.404
C01170=1057.253,-28.939,-68.351,171.155,28.834,155.405
C01171=1057.259,-28.689,-68.364,171.156,28.836,155.405
C01172=1057.266,-28.440,-68.378,171.158,28.838,155.405
C01173=1057.272,-28.191,-68.391,171.160,28.840,155.405
C01174=1057.278,-27.940,-68.404,171.161,28.842,155.406
C01175=1057.285,-27.691,-68.417,171.163,28.844,155.406
C01176=1057.291,-27.442,-68.430,171.165,28.846,155.406
C01177=1057.298,-27.192,-68.444,171.167,28.848,155.406
C01178=1057.303,-26.942,-68.458,171.168,28.849,155.406
C01179=1057.309,-26.693,-68.471,171.169,28.851,155.407
C01180=1057.315,-26.444,-68.485,171.171,28.854,155.407
C01181=1057.322,-26.194,-68.498,171.173,28.855,155.407
C01182=1057.327,-25.944,-68.511,171.174,28.858,155.407
C01183=1057.334,-25.694,-68.525,171.176,28.860,155.408
C01184=1057.340,-25.445,-68.538,171.178,28.862,155.408
C01185=1057.345,-25.195,-68.552,171.179,28.864,155.408
C01186=1057.352,-24.946,-68.565,171.181,28.866,155.408
C01187=1057.358,-24.696,-68.579,171.183,28.868,155.409
C01188=1057.364,-24.447,-68.592,171.185,28.870,155.409
C01189=1057.370,-24.197,-68.606,171.186,28.872,155.409
C01190=1057.376,-23.947,-68.620,171.188,28.874,155.409
C01191=1057.382,-23.698,-68.633,171.190,28.876,155.410
C01192=1057.389,-23.449,-68.647,171.191,28.879,155.410
C01193=1057.395,-23.198,-68.661,171.193,28.880,155.410
C01194=1057.401,-22.949,-68.674,171.194,28.882,155.410
C01195=1057.407,-22.700,-68.687,171.196,28.884,155.411
C01196=1057.413,-22.450,-68.701,171.197,28.887,155.411
C01197=1057.419,-22.200,-68.715,171.199,28.888,155.411
C01198=1057.426,-21.952,-68.729,171.201,28.890,155.411
C01199=1057.431,-21.702,-68.743,171.202,28.893,155.412
C01200=1057.438,-21.452,-68.756,171.204,28.895,155.412
C01201=1057.444,-21.203,-68.770,171.206,28.896,155.412
C01202=1057.450,-20.953,-68.783,171.208,28.899,155.412
C01203=1057.457,-20.703,-68.797,171.209,28.901,155.412
C01204=1057.462,-20.454,-68.811,171.211,28.903,155.413
C01205=1057.468,-20.204,-68.824,171.213,28.905,155.413
C01206=1057.474,-19.954,-68.838,171.214,28.907,155.413
C01207=1057.481,-19.705,-68.852,171.215,28.909,155.413
C01208=1057.487,-19.456,-68.866,171.217,28.911,155.414
C01209=1057.493,-19.206,-68.880,171.219,28.913,155.414
C01210=1057.500,-18.957,-68.893,171.220,28.915,155.414
C01211=1057.506,-18.676,-68.909,171.222,28.918,155.415
C01212=1057.513,-18.397,-68.924,171.225,28.920,155.415
C01213=1057.520,-18.116,-68.940,171.226,28.922,155.415
C01214=1057.528,-17.836,-68.955,171.228,28.925,155.415
C01215=1057.533,-17.587,-68.969,171.230,28.927,155.416
C01216=1057.540,-17.337,-68.983,171.231,28.929,155.416
C01217=1057.546,-17.088,-68.996,171.233,28.931,155.416
C01218=1057.551,-16.838,-69.010,171.235,28.933,155.416
C01219=1057.559,-16.589,-69.024,171.236,28.935,155.417
C01220=1057.564,-16.339,-69.038,171.237,28.937,155.417
C01221=1057.571,-16.089,-69.052,171.239,28.939,155.417
C01222=1057.576,-15.839,-69.066,171.241,28.941,155.417
C01223=1057.583,-15.591,-69.080,171.243,28.943,155.418
C01224=1057.590,-15.341,-69.093,171.244,28.945,155.418
C01225=1057.595,-15.091,-69.107,171.246,28.948,155.418
C01226=1057.602,-14.841,-69.121,171.248,28.950,155.418
C01227=1057.608,-14.592,-69.135,171.249,28.952,155.419
C01228=1057.613,-14.343,-69.149,171.251,28.954,155.419
C01229=1057.620,-14.093,-69.163,171.252,28.956,155.419
C01230=1057.626,-13.844,-69.177,171.254,28.958,155.419
C01231=1057.632,-13.594,-69.192,171.255,28.960,155.420
C01232=1057.638,-13.344,-69.205,171.257,28.962,155.420
C01233=1057.644,-13.095,-69.219,171.259,28.965,155.420
C01234=1057.650,-12.845,-69.234,171.260,28.967,155.420
C01235=1057.656,-12.596,-69.247,171.262,28.969,155.421
C01236=1057.663,-12.346,-69.262,171.264,28.971,155.421
C01237=1057.668,-12.097,-69.276,171.266,28.973,155.421
C01238=1057.675,-11.847,-69.290,171.267,28.976,155.422
C01239=1057.681,-11.598,-69.304,171.268,28.978,155.422
C01240=1057.686,-11.348,-69.318,171.270,28.980,155.422
C01241=1057.693,-11.099,-69.332,171.271,28.982,155.422
C01242=1057.699,-10.849,-69.346,171.273,28.984,155.423
C01243=1057.706,-10.600,-69.360,171.275,28.986,155.423
C01244=1057.711,-10.350,-69.374,171.277,28.989,155.423
C01245=1057.718,-10.101,-69.389,171.278,28.991,155.423
C01246=1057.723,-9.851,-69.403,171.280,28.993,155.424
C01247=1057.730,-9.601,-69.417,171.282,28.995,155.424
C01248=1057.736,-9.352,-69.431,171.282,28.997,155.424
C01249=1057.742,-9.102,-69.446,171.284,28.999,155.425
C01250=1057.748,-8.853,-69.460,171.286,29.002,155.425
C01251=1057.754,-8.603,-69.474,171.287,29.004,155.425
C01252=1057.760,-8.354,-69.488,171.289,29.006,155.425
C01253=1057.767,-8.104,-69.502,171.291,29.008,155.426
C01254=1057.773,-7.855,-69.517,171.293,29.010,155.426
C01255=1057.779,-7.605,-69.531,171.294,29.013,155.426
C01256=1057.785,-7.356,-69.545,171.296,29.015,155.426
C01257=1057.792,-7.106,-69.560,171.297,29.017,155.427
C01258=1057.797,-6.857,-69.574,171.298,29.019,155.427
C01259=1057.804,-6.607,-69.589,171.300,29.021,155.427
C01260=1057.810,-6.358,-69.602,171.302,29.024,155.428
C01261=1057.816,-6.108,-69.617,171.304,29.026,155.428
C01262=1057.822,-5.858,-69.631,171.305,29.028,155.428
C01263=1057.832,-5.474,-69.653,171.308,29.031,155.429
C01264=1057.841,-5.089,-69.675,171.310,29.035,155.429
C01265=1057.851,-4.705,-69.697,171.312,29.037,155.429
C01266=1057.861,-4.320,-69.719,171.315,29.041,155.430
C01267=1057.867,-4.071,-69.733,171.316,29.043,155.430
C01268=1057.873,-3.821,-69.748,171.318,29.045,155.430
C01269=1057.879,-3.572,-69.762,171.320,29.048,155.431
C01270=1057.885,-3.322,-69.777,171.321,29.050,155.431
C01271=1057.895,-2.927,-69.800,171.324,29.053,155.431
C01272=1057.904,-2.530,-69.822,171.327,29.057,155.432
C01273=1057.914,-2.133,-69.846,171.329,29.061,155.432
C01274=1057.924,-1.737,-69.869,171.332,29.064,155.433
C01275=1057.929,-1.488,-69.884,171.333,29.066,155.433
C01276=1057.936,-1.239,-69.899,171.334,29.069,155.433
C01277=1057.942,-0.988,-69.913,171.336,29.071,155.434
C01278=1057.948,-0.739,-69.928,171.337,29.073,155.434
C01279=1057.954,-0.490,-69.943,171.339,29.076,155.434
C01280=1057.960,-0.241,-69.957,171.341,29.078,155.435
C01281=1057.966,0.009,-69.971,171.343,29.080,155.435
C01282=1057.972,0.258,-69.986,171.343,29.083,155.435
C01283=1057.978,0.508,-70.001,171.345,29.085,155.436
C01284=1057.984,0.758,-70.016,171.347,29.087,155.436
C01285=1057.990,1.007,-70.030,171.348,29.089,155.436
C01286=1057.997,1.256,-70.045,171.350,29.091,155.436
C01287=1058.002,1.506,-70.059,171.352,29.094,155.437
C01288=1058.008,1.756,-70.074,171.353,29.096,155.437
C01289=1058.015,2.005,-70.089,171.354,29.098,155.437
C01290=1058.021,2.254,-70.104,171.356,29.101,155.438
C01291=1058.027,2.504,-70.119,171.358,29.103,155.438
C01292=1058.033,2.753,-70.133,171.359,29.106,155.438
C01293=1058.039,3.003,-70.148,171.361,29.108,155.439
C01294=1058.045,3.253,-70.162,171.363,29.110,155.439
C01295=1058.051,3.502,-70.177,171.364,29.112,155.439
C01296=1058.057,3.751,-70.192,171.365,29.114,155.439
C01297=1058.064,4.001,-70.207,171.367,29.117,155.440
C01298=1058.070,4.250,-70.222,171.368,29.119,155.440
C01299=1058.075,4.500,-70.237,171.370,29.121,155.440
C01300=1058.082,4.750,-70.252,171.372,29.124,155.441
C01301=1058.087,4.999,-70.267,171.374,29.126,155.441
C01302=1058.094,5.248,-70.282,171.374,29.128,155.441
C01303=1058.100,5.498,-70.296,171.376,29.131,155.442
C01304=1058.106,5.747,-70.311,171.378,29.133,155.442
C01305=1058.112,5.996,-70.326,171.379,29.135,155.442
C01306=1058.119,6.246,-70.341,171.381,29.137,155.442
C01307=1058.125,6.495,-70.356,171.383,29.140,155.443
C01308=1058.131,6.745,-70.370,171.384,29.142,155.443
C01309=1058.137,6.994,-70.385,171.385,29.144,155.443
C01310=1058.144,7.244,-70.400,171.387,29.146,155.444
C01311=1058.149,7.493,-70.415,171.389,29.148,155.444
C01312=1058.155,7.743,-70.430,171.390,29.151,155.444
C01313=1058.161,7.993,-70.445,171.392,29.153,155.445
C01314=1058.168,8.242,-70.460,171.394,29.156,155.445
C01315=1058.174,8.491,-70.475,171.395,29.158,155.445
C01316=1058.180,8.741,-70.490,171.396,29.160,155.445
C01317=1058.186,8.991,-70.505,171.398,29.163,155.446
C01318=1058.193,9.240,-70.520,171.400,29.165,155.446
C01319=1058.199,9.489,-70.534,171.401,29.167,155.446
C01320=1058.205,9.739,-70.549,171.403,29.169,155.447
C01321=1058.211,9.988,-70.564,171.404,29.171,155.447
C01322=1058.217,10.238,-70.580,171.406,29.174,155.447
C01323=1058.223,10.487,-70.594,171.407,29.176,155.448
C01324=1058.229,10.737,-70.609,171.409,29.178,155.448
C01325=1058.236,10.987,-70.624,171.411,29.181,155.448
C01326=1058.242,11.236,-70.640,171.412,29.183,155.449
C01327=1058.249,11.485,-70.655,171.413,29.185,155.449
C01328=1058.254,11.734,-70.669,171.415,29.188,155.449
C01329=1058.261,11.984,-70.684,171.417,29.190,155.449
C01330=1058.266,12.234,-70.700,171.418,29.192,155.450
C01331=1058.273,12.484,-70.715,171.420,29.195,155.450
C01332=1058.279,12.733,-70.731,171.422,29.197,155.450
C01333=1058.285,12.982,-70.745,171.422,29.199,155.451
C01334=1058.292,13.231,-70.760,171.424,29.201,155.451
C01335=1058.299,13.516,-70.777,171.426,29.204,155.451
C01336=1058.306,13.799,-70.794,171.427,29.207,155.452
C01337=1058.313,14.083,-70.812,171.429,29.209,155.452
C01338=1058.320,14.366,-70.829,171.431,29.212,155.452
C01339=1058.326,14.616,-70.844,171.432,29.214,155.453
C01340=1058.332,14.866,-70.859,171.434,29.217,155.453
C01341=1058.338,15.114,-70.875,171.436,29.219,155.453
C01342=1058.344,15.364,-70.890,171.438,29.221,155.454
C01343=1058.350,15.614,-70.905,171.439,29.224,155.454
C01344=1058.357,15.863,-70.921,171.440,29.226,155.454
C01345=1058.363,16.113,-70.936,171.442,29.228,155.455
C01346=1058.369,16.362,-70.951,171.443,29.231,155.455
C01347=1058.374,16.611,-70.966,171.445,29.233,155.455
C01348=1058.381,16.861,-70.982,171.447,29.235,155.455
C01349=1058.387,17.110,-70.997,171.448,29.238,155.456
C01350=1058.393,17.360,-71.013,171.449,29.240,155.456
C01351=1058.400,17.609,-71.028,171.451,29.242,155.456
C01352=1058.406,17.859,-71.043,171.453,29.245,155.457
C01353=1058.411,18.108,-71.058,171.454,29.247,155.457
C01354=1058.418,18.357,-71.074,171.456,29.249,155.457
C01355=1058.423,18.607,-71.090,171.457,29.252,155.458
C01356=1058.430,18.856,-71.105,171.458,29.254,155.458
C01357=1058.436,19.106,-71.120,171.460,29.256,155.458
C01358=1058.442,19.356,-71.136,171.462,29.259,155.459
C01359=1058.449,19.605,-71.151,171.464,29.261,155.459
C01360=1058.454,19.855,-71.167,171.464,29.264,155.459
C01361=1058.461,20.103,-71.182,171.466,29.266,155.460
C01362=1058.467,20.353,-71.197,171.468,29.268,155.460
C01363=1058.473,20.602,-71.213,171.469,29.271,155.460
C01364=1058.479,20.852,-71.228,171.471,29.273,155.461
C01365=1058.485,21.102,-71.244,171.472,29.276,155.461
C01366=1058.492,21.351,-71.260,171.474,29.278,155.461
C01367=1058.497,21.601,-71.275,171.475,29.280,155.462
C01368=1058.503,21.850,-71.291,171.477,29.283,155.462
C01369=1058.510,22.100,-71.306,171.479,29.285,155.462
C01370=1058.515,22.348,-71.322,171.479,29.288,155.463
C01371=1058.521,22.598,-71.337,171.481,29.290,155.463
C01372=1058.527,22.847,-71.353,171.483,29.292,155.463
C01373=1058.534,23.097,-71.368,171.484,29.295,155.464
C01374=1058.540,23.346,-71.385,171.486,29.297,155.464
C01375=1058.546,23.596,-71.400,171.487,29.299,155.464
C01376=1058.552,23.845,-71.416,171.489,29.302,155.465
C01377=1058.559,24.094,-71.431,171.490,29.304,155.465
C01378=1058.564,24.344,-71.447,171.492,29.307,155.465
C01379=1058.571,24.593,-71.463,171.494,29.309,155.466
C01380=1058.577,24.843,-71.478,171.494,29.311,155.466
C01381=1058.583,25.092,-71.494,171.496,29.314,155.466
C01382=1058.589,25.342,-71.509,171.498,29.316,155.467
C01383=1058.595,25.592,-71.526,171.500,29.318,155.467
C01384=1058.602,25.841,-71.541,171.501,29.321,155.467
C01385=1058.607,26.091,-71.557,171.502,29.323,155.468
C01386=1058.613,26.339,-71.572,171.504,29.325,155.468
C01387=1058.619,26.589,-71.588,171.505,29.328,155.468
C01388=1058.626,26.838,-71.603,171.507,29.330,155.469
C01389=1058.632,27.087,-71.620,171.509,29.333,155.469
C01390=1058.637,27.337,-71.635,171.510,29.335,155.469
C01391=1058.644,27.586,-71.651,171.511,29.337,155.470
C01392=1058.650,27.836,-71.667,171.513,29.340,155.470
C01393=1058.656,28.086,-71.682,171.515,29.342,155.470
C01394=1058.662,28.335,-71.698,171.516,29.345,155.471
C01395=1058.668,28.584,-71.715,171.517,29.347,155.471
C01396=1058.675,28.833,-71.730,171.519,29.350,155.471
C01397=1058.680,29.083,-71.746,171.521,29.352,155.472
C01398=1058.686,29.333,-71.762,171.522,29.355,155.472
C01399=1058.693,29.618,-71.780,171.524,29.357,155.472
C01400=1058.701,29.903,-71.799,171.526,29.360,155.473
C01401=1058.707,30.187,-71.817,171.527,29.363,155.473
C01402=1058.714,30.473,-71.835,171.529,29.366,155.474
C01403=1058.721,30.722,-71.851,171.531,29.368,155.474
C01404=1058.727,30.971,-71.867,171.531,29.371,155.474
C01405=1058.733,31.221,-71.883,171.533,29.373,155.475
C01406=1058.738,31.471,-71.899,171.535,29.375,155.475
C01407=1058.744,31.720,-71.915,171.536,29.378,155.475
C01408=1058.751,31.969,-71.930,171.538,29.380,155.476
C01409=1058.757,32.218,-71.947,171.539,29.382,155.476
C01410=1058.763,32.468,-71.963,171.541,29.385,155.476
C01411=1058.768,32.718,-71.979,171.542,29.387,155.477
C01412=1058.775,32.967,-71.994,171.544,29.390,155.477
C01413=1058.781,33.216,-72.010,171.546,29.392,155.477
C01414=1058.787,33.466,-72.027,171.546,29.395,155.478
C01415=1058.793,33.715,-72.043,171.548,29.397,155.478
C01416=1058.799,33.964,-72.059,171.550,29.400,155.478
C01417=1058.806,34.214,-72.075,171.552,29.402,155.479
C01418=1058.812,34.463,-72.092,171.552,29.405,155.479
C01419=1058.818,34.713,-72.107,171.554,29.407,155.479
C01420=1058.824,34.963,-72.123,171.556,29.410,155.480
C01421=1058.830,35.212,-72.140,171.557,29.412,155.480
C01422=1058.836,35.461,-72.155,171.559,29.414,155.480
C01423=1058.842,35.710,-72.171,171.560,29.416,155.481
C01424=1058.848,35.960,-72.188,171.562,29.419,155.481
C01425=1058.854,36.209,-72.204,171.563,29.422,155.482
C01426=1058.860,36.458,-72.220,171.565,29.424,155.482
C01427=1058.867,36.707,-72.236,171.566,29.427,155.482
C01428=1058.873,36.957,-72.253,171.567,29.429,155.483
C01429=1058.879,37.207,-72.269,171.569,29.432,155.483
C01430=1058.885,37.456,-72.285,171.571,29.434,155.483
C01431=1058.891,37.706,-72.301,171.572,29.437,155.484
C01432=1058.897,37.955,-72.318,171.573,29.439,155.484
C01433=1058.903,38.204,-72.334,171.575,29.441,155.484
C01434=1058.909,38.454,-72.350,171.577,29.443,155.485
C01435=1058.915,38.703,-72.366,171.578,29.446,155.485
C01436=1058.921,38.952,-72.383,171.579,29.449,155.485
C01437=1058.928,39.202,-72.399,171.581,29.451,155.486
C01438=1058.934,39.452,-72.415,171.582,29.454,155.486
C01439=1058.940,39.701,-72.432,171.584,29.456,155.486
C01440=1058.945,39.950,-72.448,171.586,29.459,155.487
C01441=1058.951,40.200,-72.464,171.587,29.461,155.487
C01442=1058.957,40.449,-72.481,171.588,29.463,155.487
C01443=1058.963,40.698,-72.497,171.590,29.466,155.488
C01444=1058.970,40.947,-72.514,171.592,29.468,155.488
C01445=1058.976,41.197,-72.530,171.592,29.471,155.489
C01446=1058.982,41.447,-72.547,171.594,29.474,155.489
C01447=1058.988,41.696,-72.563,171.596,29.476,155.489
C01448=1058.994,41.945,-72.579,171.598,29.479,155.490
C01449=1059.000,42.195,-72.595,171.599,29.481,155.490
C01450=1059.006,42.444,-72.612,171.600,29.483,155.490
C01451=1059.012,42.694,-72.628,171.602,29.486,155.491
C01452=1059.019,42.943,-72.645,171.603,29.488,155.491
C01453=1059.025,43.192,-72.661,171.605,29.491,155.491
C01454=1059.031,43.441,-72.678,171.606,29.493,155.492
C01455=1059.037,43.691,-72.694,171.608,29.496,155.492
C01456=1059.043,43.940,-72.710,171.609,29.499,155.493
C01457=1059.049,44.190,-72.728,171.611,29.501,155.493
C01458=1059.055,44.439,-72.744,171.612,29.503,155.493
C01459=1059.061,44.689,-72.761,171.613,29.506,155.494
C01460=1059.066,44.938,-72.778,171.615,29.508,155.494
C01461=1059.072,45.187,-72.795,171.617,29.511,155.494
C01462=1059.078,45.436,-72.811,171.618,29.513,155.495
C01463=1059.085,45.721,-72.830,171.620,29.516,155.495
C01464=1059.091,46.006,-72.849,171.622,29.519,155.495
C01465=1059.099,46.291,-72.868,171.624,29.523,155.496
C01466=1059.106,46.576,-72.887,171.625,29.525,155.496
C01467=1059.112,46.826,-72.904,171.626,29.528,155.497
C01468=1059.117,47.075,-72.920,171.628,29.530,155.497
C01469=1059.123,47.325,-72.937,171.629,29.533,155.497
C01470=1059.130,47.574,-72.954,171.631,29.536,155.498
C01471=1059.135,47.824,-72.971,171.632,29.538,155.498
C01472=1059.141,48.073,-72.987,171.633,29.540,155.499
C01473=1059.147,48.322,-73.004,171.635,29.543,155.499
C01474=1059.153,48.571,-73.020,171.637,29.546,155.499
C01475=1059.159,48.821,-73.038,171.638,29.548,155.500
C01476=1059.165,49.070,-73.055,171.639,29.550,155.500
C01477=1059.171,49.320,-73.071,171.641,29.553,155.500
C01478=1059.177,49.569,-73.088,171.643,29.555,155.501
C01479=1059.182,49.818,-73.105,171.643,29.558,155.501
C01480=1059.189,50.067,-73.122,171.645,29.561,155.502
C01481=1059.195,50.317,-73.138,171.647,29.563,155.502
C01482=1059.201,50.566,-73.155,171.649,29.566,155.502
C01483=1059.207,50.815,-73.172,171.650,29.568,155.503
C01484=1059.213,51.065,-73.189,171.651,29.570,155.503
C01485=1059.219,51.314,-73.206,171.653,29.573,155.503
C01486=1059.225,51.564,-73.223,171.654,29.576,155.504
C01487=1059.232,51.813,-73.240,171.656,29.579,155.504
C01488=1059.237,52.063,-73.257,171.657,29.581,155.504
C01489=1059.243,52.311,-73.274,171.659,29.583,155.505
C01490=1059.249,52.561,-73.290,171.660,29.586,155.505
C01491=1059.255,52.811,-73.307,171.662,29.588,155.506
C01492=1059.261,53.060,-73.324,171.663,29.591,155.506
C01493=1059.267,53.309,-73.340,171.664,29.594,155.506
C01494=1059.273,53.559,-73.358,171.666,29.596,155.507
C01495=1059.279,53.808,-73.375,171.668,29.598,155.507
C01496=1059.285,54.057,-73.392,171.669,29.601,155.507
C01497=1059.292,54.307,-73.409,171.670,29.603,155.508
C01498=1059.297,54.556,-73.426,171.672,29.606,155.508
C01499=1059.304,54.805,-73.443,171.674,29.609,155.509
C01500=1059.310,55.055,-73.460,171.676,29.611,155.509
C01501=1059.316,55.304,-73.477,171.676,29.613,155.509
C01502=1059.322,55.553,-73.493,171.678,29.616,155.510
C01503=1059.328,55.803,-73.511,171.680,29.618,155.510
C01504=1059.334,56.052,-73.528,171.681,29.621,155.510
C01505=1059.339,56.301,-73.545,171.682,29.624,155.511
C01506=1059.346,56.551,-73.562,171.684,29.626,155.511
C01507=1059.352,56.800,-73.578,171.686,29.629,155.511
C01508=1059.358,57.049,-73.596,171.687,29.631,155.512
C01509=1059.365,57.299,-73.613,171.688,29.633,155.512
C01510=1059.370,57.548,-73.630,171.690,29.636,155.513
C01511=1059.377,57.798,-73.648,171.691,29.639,155.513
C01512=1059.383,58.046,-73.665,171.693,29.641,155.513
C01513=1059.389,58.296,-73.681,171.695,29.644,155.514
C01514=1059.395,58.545,-73.699,171.696,29.646,155.514
C01515=1059.401,58.794,-73.716,171.697,29.648,155.514
C01516=1059.407,59.045,-73.733,171.699,29.651,155.515
C01517=1059.413,59.293,-73.750,171.701,29.653,155.515
C01518=1059.420,59.542,-73.767,171.702,29.656,155.515
C01519=1059.425,59.792,-73.784,171.703,29.659,155.516
C01520=1059.432,60.041,-73.801,171.705,29.661,155.516
C01521=1059.438,60.291,-73.819,171.707,29.663,155.517
C01522=1059.444,60.540,-73.836,171.707,29.666,155.517
C01523=1059.451,60.790,-73.853,171.709,29.668,155.517
C01524=1059.456,61.039,-73.870,171.711,29.671,155.518
C01525=1059.463,61.288,-73.888,171.713,29.674,155.518
C01526=1059.468,61.538,-73.904,171.714,29.676,155.518
C01527=1059.476,61.822,-73.924,171.716,29.679,155.519
C01528=1059.483,62.106,-73.944,171.718,29.681,155.519
C01529=1059.489,62.392,-73.963,171.719,29.685,155.520
C01530=1059.497,62.676,-73.983,171.721,29.687,155.520
C01531=1059.503,62.926,-74.001,171.722,29.689,155.520
C01532=1059.509,63.174,-74.018,171.724,29.692,155.521
C01533=1059.516,63.424,-74.035,171.725,29.695,155.521
C01534=1059.521,63.673,-74.052,171.727,29.697,155.521
C01535=1059.528,63.923,-74.069,171.729,29.700,155.522
C01536=1059.534,64.172,-74.087,171.729,29.702,155.522
C01537=1059.540,64.421,-74.104,171.731,29.704,155.523
C01538=1059.546,64.670,-74.122,171.733,29.707,155.523
C01539=1059.552,64.920,-74.140,171.735,29.710,155.523
C01540=1059.558,65.169,-74.156,171.735,29.712,155.524
C01541=1059.564,65.419,-74.174,171.737,29.715,155.524
C01542=1059.570,65.668,-74.192,171.739,29.717,155.524
C01543=1059.576,65.918,-74.209,171.740,29.720,155.525
C01544=1059.582,66.167,-74.227,171.741,29.722,155.525
C01545=1059.588,66.415,-74.244,171.743,29.725,155.526
C01546=1059.594,66.665,-74.261,171.745,29.727,155.526
C01547=1059.600,66.914,-74.279,171.746,29.730,155.526
C01548=1059.607,67.164,-74.296,171.747,29.732,155.527
C01549=1059.612,67.413,-74.314,171.749,29.735,155.527
C01550=1059.618,67.662,-74.332,171.751,29.738,155.527
C01551=1059.624,67.911,-74.349,171.752,29.740,155.528
C01552=1059.631,68.161,-74.367,171.754,29.743,155.528
C01553=1059.636,68.410,-74.384,171.755,29.745,155.529
C01554=1059.642,68.660,-74.402,171.756,29.748,155.529
C01555=1059.649,68.908,-74.419,171.758,29.750,155.529
C01556=1059.655,69.158,-74.437,171.760,29.753,155.530
C01557=1059.661,69.408,-74.455,171.761,29.755,155.530
C01558=1059.666,69.657,-74.473,171.762,29.758,155.530
C01559=1059.673,69.906,-74.490,171.764,29.760,155.531
C01560=1059.679,70.155,-74.508,171.766,29.763,155.531
C01561=1059.685,70.405,-74.526,171.767,29.765,155.532
C01562=1059.690,70.654,-74.543,171.768,29.768,155.532
C01563=1059.697,70.904,-74.561,171.770,29.771,155.532
C01564=1059.702,71.153,-74.579,171.772,29.773,155.533
C01565=1059.709,71.402,-74.596,171.773,29.776,155.533
C01566=1059.715,71.651,-74.614,171.774,29.778,155.534
C01567=1059.721,71.901,-74.632,171.776,29.781,155.534
C01568=1059.726,72.150,-74.650,171.778,29.784,155.534
C01569=1059.733,72.399,-74.668,171.779,29.786,155.535
C01570=1059.738,72.648,-74.685,171.780,29.788,155.535
C01571=1059.744,72.898,-74.703,171.782,29.791,155.535
C01572=1059.751,73.148,-74.720,171.784,29.794,155.536
C01573=1059.757,73.396,-74.739,171.785,29.797,155.536
C01574=1059.763,73.646,-74.757,171.786,29.799,155.537
C01575=1059.768,73.895,-74.774,171.788,29.801,155.537
C01576=1059.775,74.144,-74.792,171.789,29.804,155.537
C01577=1059.780,74.393,-74.810,171.791,29.807,155.538
C01578=1059.786,74.643,-74.828,171.793,29.809,155.538
C01579=1059.793,74.892,-74.846,171.794,29.812,155.538
C01580=1059.798,75.141,-74.864,171.795,29.814,155.539
C01581=1059.805,75.391,-74.881,171.797,29.817,155.539
C01582=1059.811,75.640,-74.899,171.799,29.820,155.540
C01583=1059.817,75.889,-74.917,171.800,29.822,155.540
C01584=1059.823,76.139,-74.935,171.801,29.824,155.540
C01585=1059.829,76.388,-74.953,171.803,29.827,155.541
C01586=1059.835,76.638,-74.971,171.805,29.830,155.541
C01587=1059.841,76.886,-74.989,171.806,29.832,155.541
C01588=1059.847,77.136,-75.007,171.807,29.835,155.542
C01589=1059.853,77.385,-75.025,171.809,29.837,155.542
C01590=1059.859,77.634,-75.043,171.811,29.840,155.543
C01591=1059.866,77.919,-75.064,171.812,29.843,155.543
C01592=1059.873,78.204,-75.084,171.814,29.845,155.543
C01593=1059.879,78.488,-75.105,171.816,29.849,155.544
C01594=1059.886,78.772,-75.126,171.817,29.852,155.544
C01595=1059.892,79.022,-75.144,171.819,29.854,155.545
C01596=1059.898,79.271,-75.161,171.820,29.857,155.545
C01597=1059.904,79.520,-75.180,171.822,29.860,155.546
C01598=1059.910,79.770,-75.198,171.823,29.862,155.546
C01599=1059.916,80.018,-75.216,171.825,29.864,155.546
C01600=1059.922,80.268,-75.234,171.827,29.867,155.547
C01601=1059.927,80.517,-75.252,171.828,29.870,155.547
C01602=1059.934,80.767,-75.271,171.829,29.872,155.548
C01603=1059.940,81.016,-75.289,171.831,29.875,155.548
C01604=1059.946,81.265,-75.307,171.833,29.878,155.548
C01605=1059.952,81.514,-75.325,171.833,29.880,155.549
C01606=1059.958,81.764,-75.344,171.835,29.883,155.549
C01607=1059.963,82.013,-75.362,171.837,29.885,155.549
C01608=1059.969,82.262,-75.380,171.839,29.888,155.550
C01609=1059.975,82.512,-75.398,171.839,29.891,155.550
C01610=1059.981,82.760,-75.417,171.841,29.893,155.551
C01611=1059.987,83.010,-75.434,171.843,29.896,155.551
C01612=1059.994,83.259,-75.453,171.845,29.899,155.552
C01613=1059.999,83.508,-75.471,171.846,29.901,155.552
C01614=1060.005,83.758,-75.490,171.847,29.903,155.552
C01615=1060.011,84.007,-75.508,171.849,29.906,155.553
C01616=1060.017,84.256,-75.526,171.851,29.909,155.553
C01617=1060.023,84.505,-75.544,171.852,29.912,155.553
C01618=1060.029,84.755,-75.563,171.853,29.914,155.554
C01619=1060.035,85.005,-75.581,171.855,29.916,155.554
C01620=1060.041,85.253,-75.600,171.856,29.919,155.555
C01621=1060.047,85.503,-75.617,171.858,29.922,155.555
C01622=1060.053,85.752,-75.636,171.860,29.924,155.555
C01623=1060.059,86.000,-75.654,171.861,29.927,155.556
C01624=1060.064,86.250,-75.673,171.862,29.929,155.556
C01625=1060.071,86.500,-75.692,171.864,29.932,155.557
C01626=1060.077,86.749,-75.710,171.866,29.934,155.557
C01627=1060.083,86.998,-75.728,171.868,29.937,155.557
C01628=1060.089,87.247,-75.746,171.868,29.940,155.558
C01629=1060.095,87.497,-75.765,171.870,29.942,155.558
C01630=1060.101,87.746,-75.784,171.872,29.945,155.558
C01631=1060.107,87.995,-75.802,171.874,29.947,155.559
C01632=1060.113,88.244,-75.820,171.875,29.950,155.559
C01633=1060.119,88.493,-75.838,171.876,29.953,155.560
C01634=1060.125,88.743,-75.858,171.878,29.955,155.560
C01635=1060.131,88.992,-75.876,171.880,29.957,155.560
C01636=1060.137,89.241,-75.894,171.881,29.960,155.561
C01637=1060.143,89.490,-75.913,171.882,29.963,155.561
C01638=1060.150,89.740,-75.931,171.884,29.965,155.562
C01639=1060.155,89.989,-75.950,171.886,29.968,155.562
C01640=1060.162,90.238,-75.968,171.887,29.970,155.562
C01641=1060.168,90.488,-75.986,171.889,29.973,155.563
C01642=1060.174,90.736,-76.005,171.890,29.976,155.563
C01643=1060.179,90.986,-76.024,171.891,29.978,155.564
C01644=1060.186,91.235,-76.043,171.893,29.981,155.564
C01645=1060.191,91.484,-76.062,171.895,29.984,155.564
C01646=1060.197,91.733,-76.079,171.897,29.986,155.565
C01647=1060.203,91.983,-76.099,171.897,29.988,155.565
C01648=1060.209,92.232,-76.117,171.899,29.991,155.565
C01649=1060.215,92.481,-76.136,171.901,29.994,155.566
C01650=1060.221,92.731,-76.155,171.903,29.996,155.566
C01651=1060.226,92.980,-76.173,171.904,29.999,155.567
C01652=1060.232,93.229,-76.192,171.905,30.002,155.567
C01653=1060.239,93.478,-76.211,171.907,30.004,155.568
C01654=1060.245,93.728,-76.230,171.909,30.007,155.568
C01655=1060.251,94.012,-76.251,171.910,30.010,155.568
C01656=1060.258,94.297,-76.273,171.912,30.013,155.569
C01657=1060.265,94.581,-76.294,171.914,30.016,155.569
C01658=1060.272,94.865,-76.315,171.915,30.019,155.570
C01659=1060.277,95.115,-76.334,171.917,30.021,155.570
C01660=1060.283,95.364,-76.353,171.919,30.024,155.570
C01661=1060.289,95.613,-76.372,171.921,30.027,155.571
C01662=1060.295,95.863,-76.391,171.921,30.029,155.571
C01663=1060.301,96.112,-76.410,171.923,30.032,155.572
C01664=1060.308,96.361,-76.428,171.925,30.035,155.572
C01665=1060.313,96.610,-76.447,171.927,30.037,155.572
C01666=1060.319,96.859,-76.466,171.928,30.040,155.573
C01667=1060.325,97.108,-76.485,171.929,30.042,155.573
C01668=1060.331,97.357,-76.504,171.931,30.045,155.574
C01669=1060.337,97.607,-76.523,171.933,30.048,155.574
C01670=1060.343,97.856,-76.542,171.934,30.050,155.574
C01671=1060.349,98.105,-76.561,171.936,30.053,155.575
C01672=1060.355,98.355,-76.580,171.937,30.055,155.575
C01673=1060.361,98.604,-76.599,171.939,30.058,155.576
C01674=1060.368,98.853,-76.617,171.940,30.060,155.576
C01675=1060.373,99.102,-76.636,171.942,30.063,155.576
C01676=1060.379,99.351,-76.655,171.944,30.066,155.577
C01677=1060.385,99.600,-76.674,171.945,30.068,155.577
C01678=1060.391,99.850,-76.693,171.946,30.071,155.578
C01679=1060.397,100.099,-76.712,171.948,30.074,155.578
C01680=1060.403,100.348,-76.731,171.950,30.076,155.578
C01681=1060.409,100.598,-76.750,171.952,30.079,155.579
C01682=1060.415,100.847,-76.769,171.953,30.081,155.579
C01683=1060.421,101.095,-76.789,171.954,30.084,155.580
C01684=1060.427,101.345,-76.808,171.956,30.086,155.580
C01685=1060.433,101.594,-76.827,171.957,30.089,155.580
C01686=1060.439,101.843,-76.846,171.959,30.092,155.581
C01687=1060.445,102.093,-76.865,171.961,30.095,155.581
C01688=1060.451,102.342,-76.884,171.962,30.097,155.582
C01689=1060.456,102.591,-76.903,171.963,30.100,155.582
C01690=1060.462,102.840,-76.923,171.965,30.103,155.582
C01691=1060.468,103.089,-76.942,171.967,30.105,155.583
C01692=1060.474,103.338,-76.961,171.969,30.107,155.583
C01693=1060.479,103.588,-76.980,171.970,30.110,155.584
C01694=1060.486,103.837,-76.999,171.971,30.113,155.584
C01695=1060.492,104.086,-77.019,171.973,30.115,155.584
C01696=1060.498,104.335,-77.038,171.975,30.118,155.585
C01697=1060.503,104.585,-77.057,171.976,30.121,155.585
C01698=1060.509,104.834,-77.077,171.978,30.123,155.586
C01699=1060.515,105.083,-77.095,171.979,30.126,155.586
C01700=1060.521,105.332,-77.115,171.981,30.129,155.586
C01701=1060.527,105.581,-77.134,171.982,30.131,155.587
C01702=1060.533,105.831,-77.154,171.984,30.134,155.587
C01703=1060.539,106.079,-77.173,171.986,30.137,155.588
C01704=1060.545,106.329,-77.192,171.988,30.139,155.588
C01705=1060.551,106.578,-77.212,171.988,30.142,155.588
C01706=1060.557,106.828,-77.231,171.990,30.144,155.589
C01707=1060.563,107.077,-77.251,171.992,30.147,155.589
C01708=1060.569,107.326,-77.269,171.994,30.149,155.590
C01709=1060.575,107.575,-77.289,171.995,30.152,155.590
C01710=1060.581,107.824,-77.309,171.997,30.155,155.590
C01711=1060.586,108.073,-77.328,171.998,30.157,155.591
C01712=1060.592,108.323,-77.347,172.000,30.160,155.591
C01713=1060.599,108.571,-77.366,172.001,30.163,155.592
C01714=1060.604,108.821,-77.386,172.003,30.166,155.592
C01715=1060.610,109.069,-77.406,172.005,30.168,155.592
C01716=1060.616,109.319,-77.425,172.007,30.170,155.593
C01717=1060.622,109.568,-77.444,172.007,30.173,155.593
C01718=1060.629,109.817,-77.463,172.009,30.176,155.594
C01719=1060.635,110.102,-77.485,172.011,30.179,155.594
C01720=1060.643,110.386,-77.508,172.014,30.182,155.594
C01721=1060.648,110.671,-77.530,172.015,30.184,155.595
C01722=1060.655,110.955,-77.553,172.017,30.188,155.595
C01723=1060.662,111.204,-77.572,172.019,30.190,155.596
C01724=1060.668,111.453,-77.592,172.020,30.193,155.596
C01725=1060.673,111.703,-77.611,172.021,30.196,155.597
C01726=1060.680,111.952,-77.631,172.023,30.198,155.597
C01727=1060.686,112.201,-77.650,172.025,30.201,155.597
C01728=1060.692,112.450,-77.670,172.027,30.203,155.598
C01729=1060.697,112.700,-77.690,172.028,30.206,155.598
C01730=1060.703,112.949,-77.710,172.030,30.209,155.599
C01731=1060.709,113.198,-77.729,172.031,30.211,155.599
C01732=1060.715,113.447,-77.749,172.033,30.214,155.599
C01733=1060.721,113.696,-77.768,172.034,30.216,155.600
C01734=1060.727,113.945,-77.788,172.036,30.219,155.600
C01735=1060.732,114.194,-77.807,172.038,30.222,155.601
C01736=1060.738,114.443,-77.827,172.040,30.225,155.601
C01737=1060.744,114.693,-77.846,172.041,30.227,155.601
C01738=1060.749,114.942,-77.867,172.042,30.230,155.602
C01739=1060.756,115.191,-77.887,172.044,30.232,155.602
C01740=1060.762,115.441,-77.907,172.046,30.235,155.603
C01741=1060.767,115.690,-77.927,172.047,30.238,155.603
C01742=1060.773,115.938,-77.947,172.049,30.241,155.604
C01743=1060.778,116.188,-77.966,172.051,30.243,155.604
C01744=1060.784,116.437,-77.986,172.052,30.246,155.604
C01745=1060.790,116.686,-78.006,172.053,30.248,155.605
C01746=1060.796,116.935,-78.026,172.055,30.251,155.605
C01747=1060.802,117.184,-78.045,172.057,30.254,155.606
C01748=1060.807,117.433,-78.066,172.059,30.257,155.606
C01749=1060.813,117.683,-78.085,172.060,30.260,155.607
C01750=1060.819,117.931,-78.105,172.062,30.263,155.607
C01751=1060.826,118.181,-78.126,172.063,30.265,155.607
C01752=1060.831,118.430,-78.145,172.065,30.268,155.608
C01753=1060.837,118.679,-78.165,172.066,30.270,155.608
C01754=1060.843,118.928,-78.185,172.068,30.273,155.609
C01755=1060.849,119.177,-78.205,172.070,30.276,155.609
C01756=1060.854,119.427,-78.225,172.072,30.279,155.609
C01757=1060.860,119.676,-78.245,172.073,30.281,155.610
C01758=1060.866,119.925,-78.265,172.075,30.284,155.610
C01759=1060.872,120.174,-78.285,172.076,30.286,155.611
C01760=1060.878,120.423,-78.305,172.078,30.289,155.611
C01761=1060.883,120.673,-78.325,172.079,30.292,155.611
C01762=1060.889,120.921,-78.345,172.081,30.294,155.612
C01763=1060.895,121.170,-78.365,172.083,30.297,155.612
C01764=1060.902,121.420,-78.385,172.085,30.300,155.613
C01765=1060.907,121.669,-78.406,172.086,30.303,155.613
C01766=1060.913,121.918,-78.426,172.088,30.305,155.614
C01767=1060.919,122.167,-78.445,172.089,30.308,155.614
C01768=1060.925,122.416,-78.465,172.091,30.310,155.614
C01769=1060.930,122.666,-78.486,172.092,30.313,155.615
C01770=1060.936,122.914,-78.506,172.094,30.316,155.615
C01771=1060.942,123.163,-78.526,172.096,30.319,155.616
C01772=1060.948,123.412,-78.546,172.098,30.321,155.616
C01773=1060.954,123.661,-78.566,172.099,30.324,155.616
C01774=1060.960,123.911,-78.587,172.101,30.326,155.617
C01775=1060.966,124.160,-78.607,172.103,30.329,155.617
C01776=1060.972,124.409,-78.626,172.104,30.331,155.618
C01777=1060.977,124.658,-78.647,172.106,30.334,155.618
C01778=1060.984,124.908,-78.667,172.107,30.337,155.618
C01779=1060.990,125.156,-78.687,172.109,30.339,155.619
C01780=1060.995,125.406,-78.707,172.111,30.342,155.619
C01781=1061.001,125.654,-78.727,172.113,30.345,155.620
C01782=1061.008,125.904,-78.748,172.114,30.347,155.620
C01783=1061.014,126.189,-78.771,172.116,30.351,155.621
C01784=1061.021,126.472,-78.794,172.118,30.353,155.621
C01785=1061.028,126.757,-78.818,172.120,30.357,155.621
C01786=1061.035,127.041,-78.840,172.122,30.359,155.622
C01787=1061.040,127.290,-78.861,172.123,30.362,155.622
C01788=1061.046,127.539,-78.881,172.125,30.365,155.623
C01789=1061.053,127.789,-78.901,172.127,30.367,155.623
C01790=1061.058,128.038,-78.922,172.128,30.370,155.624
C01791=1061.064,128.287,-78.942,172.130,30.373,155.624
C01792=1061.071,128.536,-78.962,172.132,30.375,155.624
C01793=1061.076,128.785,-78.983,172.134,30.378,155.625
C01794=1061.082,129.034,-79.003,172.135,30.381,155.625
C01795=1061.089,129.284,-79.023,172.137,30.383,155.626
C01796=1061.094,129.532,-79.044,172.139,30.386,155.626
C01797=1061.100,129.781,-79.064,172.141,30.389,155.626
C01798=1061.107,130.031,-79.084,172.142,30.391,155.627
C01799=1061.112,130.280,-79.105,172.144,30.394,155.627
C01800=1061.118,130.528,-79.125,172.145,30.396,155.628
C01801=1061.125,130.778,-79.145,172.147,30.399,155.628
C01802=1061.130,131.027,-79.166,172.149,30.401,155.628
C01803=1061.136,131.277,-79.186,172.150,30.404,155.629
C01804=1061.143,131.525,-79.207,172.152,30.407,155.629
C01805=1061.148,131.774,-79.227,172.154,30.409,155.630
C01806=1061.155,132.023,-79.248,172.156,30.412,155.630
C01807=1061.160,132.273,-79.268,172.157,30.415,155.630
C01808=1061.166,132.521,-79.289,172.159,30.418,155.631
C01809=1061.172,132.771,-79.310,172.161,30.420,155.631
C01810=1061.177,133.020,-79.330,172.163,30.423,155.632
C01811=1061.183,133.269,-79.350,172.164,30.426,155.632
C01812=1061.189,133.518,-79.372,172.166,30.428,155.632
C01813=1061.195,133.767,-79.392,172.168,30.431,155.633
C01814=1061.201,134.016,-79.412,172.170,30.434,155.633
C01815=1061.207,134.266,-79.433,172.171,30.436,155.634
C01816=1061.213,134.514,-79.454,172.172,30.439,155.634
C01817=1061.219,134.764,-79.475,172.174,30.441,155.635
C01818=1061.225,135.012,-79.495,172.176,30.444,155.635
C01819=1061.230,135.261,-79.516,172.178,30.447,155.635
